};
P[388]{
   GP1:
	UF : 0, UT : 6,		CONFIG : 'N U T, 0, 0, 0',
	X =  173.893  mm,	Y =   -630.176  mm,	Z =   -253.833  mm,
	W =  90.000 deg,	P =   0.000 deg,	R =   90.000 deg
};
P[389]{
   GP1:
	UF : 0, UT : 6,		CONFIG : 'N U T, 0, 0, 0',
	X =  177.098  mm,	Y =   -628.334  mm,	Z =   -253.813  mm,
	W =  90.000 deg,	P =   0.000 deg,	R =   90.000 deg
};
P[390]{
   GP1:
	UF : 0, UT : 6,		CONFIG : 'N U T, 0, 0, 0',
	X =  178.651  mm,	Y =   -627.382  mm,	Z =   -253.947  mm,
	W =  90.000 deg,	P =   0.000 deg,	R =   90.000 deg
};
P[391]{
   GP1:
	UF : 0, UT : 6,		CONFIG : 'N U T, 0, 0, 0',
	X =  180.197  mm,	Y =   -626.528  mm,	Z =   -253.855  mm,
	W =  90.000 deg,	P =   0.000 deg,	R =   90.000 deg
};
P[392]{
   GP1:
	UF : 0, UT : 6,		CONFIG : 'N U T, 0, 0, 0',
	X =  180.887  mm,	Y =   -626.108  mm,	Z =   -253.906  mm,
	W =  90.000 deg,	P =   0.000 deg,	R =   90.000 deg
};
P[393]{
   GP1:
	UF : 0, UT : 6,		CONFIG : 'N U T, 0, 0, 0',
	X =  181.456  mm,	Y =   -625.692  mm,	Z =   -254.117  mm,
	W =  90.000 deg,	P =   0.000 deg,	R =   90.000 deg
};
P[394]{
   GP1:
	UF : 0, UT : 6,		CONFIG : 'N U T, 0, 0, 0',
	X =  182.165  mm,	Y =   -625.424  mm,	Z =   -253.772  mm,
	W =  90.000 deg,	P =   0.000 deg,	R =   90.000 deg
};
P[395]{
   GP1:
	UF : 0, UT : 6,		CONFIG : 'N U T, 0, 0, 0',
	X =  184.178  mm,	Y =   -624.237  mm,	Z =   -253.834  mm,
	W =  90.000 deg,	P =   0.000 deg,	R =   90.000 deg
};
P[396]{
   GP1:
	UF : 0, UT : 6,		CONFIG : 'N U T, 0, 0, 0',
	X =  185.737  mm,	Y =   -623.407  mm,	Z =   -253.665  mm,
	W =  90.000 deg,	P =   0.000 deg,	R =   90.000 deg
};
P[397]{
   GP1:
	UF : 0, UT : 6,		CONFIG : 'N U T, 0, 0, 0',
	X =  187.493  mm,	Y =   -622.385  mm,	Z =   -253.683  mm,
	W =  90.000 deg,	P =   0.000 deg,	R =   90.000 deg
};
P[398]{
   GP1:
	UF : 0, UT : 6,		CONFIG : 'N U T, 0, 0, 0',
	X =  188.774  mm,	Y =   -621.575  mm,	Z =   -253.856  mm,
	W =  90.000 deg,	P =   0.000 deg,	R =   90.000 deg
};
P[399]{
   GP1:
	UF : 0, UT : 6,		CONFIG : 'N U T, 0, 0, 0',
	X =  190.507  mm,	Y =   -620.610  mm,	Z =   -253.768  mm,
	W =  90.000 deg,	P =   0.000 deg,	R =   90.000 deg
};
P[400]{
   GP1:
	UF : 0, UT : 6,		CONFIG : 'N U T, 0, 0, 0',
	X =  191.557  mm,	Y =   -619.888  mm,	Z =   -254.049  mm,
	W =  90.000 deg,	P =   0.000 deg,	R =   90.000 deg
};
P[401]{
   GP1:
	UF : 0, UT : 6,		CONFIG : 'N U T, 0, 0, 0',
	X =  192.194  mm,	Y =   -619.679  mm,	Z =   -253.663  mm,
	W =  90.000 deg,	P =   0.000 deg,	R =   90.000 deg
};
P[402]{
   GP1:
	UF : 0, UT : 6,		CONFIG : 'N U T, 0, 0, 0',
	X =  193.971  mm,	Y =   -618.550  mm,	Z =   -253.914  mm,
	W =  90.000 deg,	P =   0.000 deg,	R =   90.000 deg
};
P[403]{
   GP1:
	UF : 0, UT : 6,		CONFIG : 'N U T, 0, 0, 0',
	X =  194.982  mm,	Y =   -617.974  mm,	Z =   -253.896  mm,
	W =  90.000 deg,	P =   0.000 deg,	R =   90.000 deg
};
P[404]{
   GP1:
	UF : 0, UT : 6,		CONFIG : 'N U T, 0, 0, 0',
	X =  196.361  mm,	Y =   -617.195  mm,	Z =   -253.854  mm,
	W =  90.000 deg,	P =   0.000 deg,	R =   90.000 deg
};
P[405]{
   GP1:
	UF : 0, UT : 6,		CONFIG : 'N U T, 0, 0, 0',
	X =  197.401  mm,	Y =   -616.488  mm,	Z =   -254.111  mm,
	W =  90.000 deg,	P =   0.000 deg,	R =   90.000 deg
};
P[406]{
   GP1:
	UF : 0, UT : 6,		CONFIG : 'N U T, 0, 0, 0',
	X =  198.586  mm,	Y =   -615.883  mm,	Z =   -253.918  mm,
	W =  90.000 deg,	P =   0.000 deg,	R =   90.000 deg
};
P[407]{
   GP1:
	UF : 0, UT : 6,		CONFIG : 'N U T, 0, 0, 0',
	X =  200.043  mm,	Y =   -615.098  mm,	Z =   -253.782  mm,
	W =  90.000 deg,	P =   0.000 deg,	R =   90.000 deg
};
P[408]{
   GP1:
	UF : 0, UT : 6,		CONFIG : 'N U T, 0, 0, 0',
	X =  200.867  mm,	Y =   -614.662  mm,	Z =   -253.686  mm,
	W =  90.000 deg,	P =   0.000 deg,	R =   90.000 deg
};
P[409]{
   GP1:
	UF : 0, UT : 6,		CONFIG : 'N U T, 0, 0, 0',
	X =  203.321  mm,	Y =   -613.136  mm,	Z =   -253.950  mm,
	W =  90.000 deg,	P =   0.000 deg,	R =   90.000 deg
};
P[410]{
   GP1:
	UF : 0, UT : 6,		CONFIG : 'N U T, 0, 0, 0',
	X =  204.899  mm,	Y =   -612.164  mm,	Z =   -254.098  mm,
	W =  90.000 deg,	P =   0.000 deg,	R =   90.000 deg
};
P[411]{
   GP1:
	UF : 0, UT : 6,		CONFIG : 'N U T, 0, 0, 0',
	X =  206.618  mm,	Y =   -611.234  mm,	Z =   -253.947  mm,
	W =  90.000 deg,	P =   0.000 deg,	R =   90.000 deg
};
P[412]{
   GP1:
	UF : 0, UT : 6,		CONFIG : 'N U T, 0, 0, 0',
	X =  208.390  mm,	Y =   -610.150  mm,	Z =   -254.093  mm,
	W =  90.000 deg,	P =   0.000 deg,	R =   90.000 deg
};
P[413]{
   GP1:
	UF : 0, UT : 6,		CONFIG : 'N U T, 0, 0, 0',
	X =  209.057  mm,	Y =   -609.766  mm,	Z =   -254.091  mm,
	W =  90.000 deg,	P =   0.000 deg,	R =   90.000 deg
};
P[414]{
   GP1:
	UF : 0, UT : 6,		CONFIG : 'N U T, 0, 0, 0',
	X =  210.367  mm,	Y =   -609.174  mm,	Z =   -253.692  mm,
	W =  90.000 deg,	P =   0.000 deg,	R =   90.000 deg
};
P[415]{
   GP1:
	UF : 0, UT : 6,		CONFIG : 'N U T, 0, 0, 0',
	X =  211.415  mm,	Y =   -608.428  mm,	Z =   -254.033  mm,
	W =  90.000 deg,	P =   0.000 deg,	R =   90.000 deg
};
P[416]{
   GP1:
	UF : 0, UT : 6,		CONFIG : 'N U T, 0, 0, 0',
	X =  212.531  mm,	Y =   -607.864  mm,	Z =   -253.839  mm,
	W =  90.000 deg,	P =   0.000 deg,	R =   90.000 deg
};
P[417]{
   GP1:
	UF : 0, UT : 6,		CONFIG : 'N U T, 0, 0, 0',
	X =  216.353  mm,	Y =   -605.647  mm,	Z =   -253.865  mm,
	W =  90.000 deg,	P =   0.000 deg,	R =   90.000 deg
};
P[418]{
   GP1:
	UF : 0, UT : 6,		CONFIG : 'N U T, 0, 0, 0',
	X =  217.171  mm,	Y =   -605.129  mm,	Z =   -253.976  mm,
	W =  90.000 deg,	P =   0.000 deg,	R =   90.000 deg
};
P[419]{
   GP1:
	UF : 0, UT : 6,		CONFIG : 'N U T, 0, 0, 0',
	X =  220.039  mm,	Y =   -603.422  mm,	Z =   -254.099  mm,
	W =  90.000 deg,	P =   0.000 deg,	R =   90.000 deg
};
P[420]{
   GP1:
	UF : 0, UT : 6,		CONFIG : 'N U T, 0, 0, 0',
	X =  222.534  mm,	Y =   -601.991  mm,	Z =   -254.077  mm,
	W =  90.000 deg,	P =   0.000 deg,	R =   90.000 deg
};
P[421]{
   GP1:
	UF : 0, UT : 6,		CONFIG : 'N U T, 0, 0, 0',
	X =  223.322  mm,	Y =   -601.645  mm,	Z =   -253.810  mm,
	W =  90.000 deg,	P =   0.000 deg,	R =   90.000 deg
};
P[422]{
   GP1:
	UF : 0, UT : 6,		CONFIG : 'N U T, 0, 0, 0',
	X =  226.177  mm,	Y =   -599.995  mm,	Z =   -253.815  mm,
	W =  90.000 deg,	P =   0.000 deg,	R =   90.000 deg
};
P[423]{
   GP1:
	UF : 0, UT : 6,		CONFIG : 'N U T, 0, 0, 0',
	X =  230.315  mm,	Y =   -597.495  mm,	Z =   -254.084  mm,
	W =  90.000 deg,	P =   0.000 deg,	R =   90.000 deg
};
P[424]{
   GP1:
	UF : 0, UT : 6,		CONFIG : 'N U T, 0, 0, 0',
	X =  233.160  mm,	Y =   -595.945  mm,	Z =   -253.857  mm,
	W =  90.000 deg,	P =   0.000 deg,	R =   90.000 deg
};
P[425]{
   GP1:
	UF : 0, UT : 6,		CONFIG : 'N U T, 0, 0, 0',
	X =  233.779  mm,	Y =   -595.666  mm,	Z =   -253.669  mm,
	W =  90.000 deg,	P =   0.000 deg,	R =   90.000 deg
};
P[426]{
   GP1:
	UF : 0, UT : 6,		CONFIG : 'N U T, 0, 0, 0',
	X =  235.720  mm,	Y =   -594.384  mm,	Z =   -254.058  mm,
	W =  90.000 deg,	P =   0.000 deg,	R =   90.000 deg
};
P[427]{
   GP1:
	UF : 0, UT : 6,		CONFIG : 'N U T, 0, 0, 0',
	X =  239.909  mm,	Y =   -592.111  mm,	Z =   -253.707  mm,
	W =  90.000 deg,	P =   0.000 deg,	R =   90.000 deg
};
P[428]{
   GP1:
	UF : 0, UT : 6,		CONFIG : 'N U T, 0, 0, 0',
	X =  240.586  mm,	Y =   -591.645  mm,	Z =   -253.890  mm,
	W =  90.000 deg,	P =   0.000 deg,	R =   90.000 deg
};
P[429]{
   GP1:
	UF : 0, UT : 6,		CONFIG : 'N U T, 0, 0, 0',
	X =  241.630  mm,	Y =   -591.052  mm,	Z =   -253.864  mm,
	W =  90.000 deg,	P =   0.000 deg,	R =   90.000 deg
};
P[430]{
   GP1:
	UF : 0, UT : 6,		CONFIG : 'N U T, 0, 0, 0',
	X =  243.410  mm,	Y =   -590.078  mm,	Z =   -253.734  mm,
	W =  90.000 deg,	P =   0.000 deg,	R =   90.000 deg
};
P[431]{
   GP1:
	UF : 0, UT : 6,		CONFIG : 'N U T, 0, 0, 0',
	X =  244.625  mm,	Y =   -589.217  mm,	Z =   -254.121  mm,
	W =  90.000 deg,	P =   0.000 deg,	R =   90.000 deg
};
P[432]{
   GP1:
	UF : 0, UT : 6,		CONFIG : 'N U T, 0, 0, 0',
	X =  247.372  mm,	Y =   -587.776  mm,	Z =   -253.768  mm,
	W =  90.000 deg,	P =   0.000 deg,	R =   90.000 deg
};
P[433]{
   GP1:
	UF : 0, UT : 6,		CONFIG : 'N U T, 0, 0, 0',
	X =  249.854  mm,	Y =   -586.285  mm,	Z =   -253.910  mm,
	W =  90.000 deg,	P =   0.000 deg,	R =   90.000 deg
};
P[434]{
   GP1:
	UF : 0, UT : 6,		CONFIG : 'N U T, 0, 0, 0',
	X =  252.767  mm,	Y =   -584.575  mm,	Z =   -253.975  mm,
	W =  90.000 deg,	P =   0.000 deg,	R =   90.000 deg
};
P[435]{
   GP1:
	UF : 0, UT : 6,		CONFIG : 'N U T, 0, 0, 0',
	X =  256.146  mm,	Y =   -582.657  mm,	Z =   -253.897  mm,
	W =  90.000 deg,	P =   0.000 deg,	R =   90.000 deg
};
P[436]{
   GP1:
	UF : 0, UT : 6,		CONFIG : 'N U T, 0, 0, 0',
	X =  256.773  mm,	Y =   -582.393  mm,	Z =   -253.661  mm,
	W =  90.000 deg,	P =   0.000 deg,	R =   90.000 deg
};
P[437]{
   GP1:
	UF : 0, UT : 6,		CONFIG : 'N U T, 0, 0, 0',
	X =  260.094  mm,	Y =   -580.358  mm,	Z =   -253.944  mm,
	W =  90.000 deg,	P =   0.000 deg,	R =   90.000 deg
};
P[438]{
   GP1:
	UF : 0, UT : 6,		CONFIG : 'N U T, 0, 0, 0',
	X =  261.050  mm,	Y =   -579.846  mm,	Z =   -253.849  mm,
	W =  90.000 deg,	P =   0.000 deg,	R =   90.000 deg
};
P[439]{
   GP1:
	UF : 0, UT : 6,		CONFIG : 'N U T, 0, 0, 0',
	X =  262.708  mm,	Y =   -578.893  mm,	Z =   -253.836  mm,
	W =  90.000 deg,	P =   0.000 deg,	R =   90.000 deg
};
P[440]{
   GP1:
	UF : 0, UT : 6,		CONFIG : 'N U T, 0, 0, 0',
	X =  263.927  mm,	Y =   -578.207  mm,	Z =   -253.795  mm,
	W =  90.000 deg,	P =   0.000 deg,	R =   90.000 deg
};
P[441]{
   GP1:
	UF : 0, UT : 6,		CONFIG : 'N U T, 0, 0, 0',
	X =  265.115  mm,	Y =   -577.452  mm,	Z =   -253.964  mm,
	W =  90.000 deg,	P =   0.000 deg,	R =   90.000 deg
};
P[442]{
   GP1:
	UF : 0, UT : 6,		CONFIG : 'N U T, 0, 0, 0',
	X =  265.815  mm,	Y =   -577.128  mm,	Z =   -253.767  mm,
	W =  90.000 deg,	P =   0.000 deg,	R =   90.000 deg
};
P[443]{
   GP1:
	UF : 0, UT : 6,		CONFIG : 'N U T, 0, 0, 0',
	X =  266.400  mm,	Y =   -576.646  mm,	Z =   -254.119  mm,
	W =  90.000 deg,	P =   0.000 deg,	R =   90.000 deg
};
P[444]{
   GP1:
	UF : 0, UT : 6,		CONFIG : 'N U T, 0, 0, 0',
	X =  269.651  mm,	Y =   -574.901  mm,	Z =   -253.796  mm,
	W =  90.000 deg,	P =   0.000 deg,	R =   90.000 deg
};
P[445]{
   GP1:
	UF : 0, UT : 6,		CONFIG : 'N U T, 0, 0, 0',
	X =  270.217  mm,	Y =   -574.487  mm,	Z =   -254.009  mm,
	W =  90.000 deg,	P =   0.000 deg,	R =   90.000 deg
};
P[446]{
   GP1:
	UF : 0, UT : 6,		CONFIG : 'N U T, 0, 0, 0',
	X =  270.803  mm,	Y =   -574.109  mm,	Z =   -254.105  mm,
	W =  90.000 deg,	P =   0.000 deg,	R =   90.000 deg
};
P[447]{
   GP1:
	UF : 0, UT : 6,		CONFIG : 'N U T, 0, 0, 0',
	X =  271.415  mm,	Y =   -573.808  mm,	Z =   -253.978  mm,
	W =  90.000 deg,	P =   0.000 deg,	R =   90.000 deg
};
P[448]{
   GP1:
	UF : 0, UT : 6,		CONFIG : 'N U T, 0, 0, 0',
	X =  272.339  mm,	Y =   -573.365  mm,	Z =   -253.756  mm,
	W =  90.000 deg,	P =   0.000 deg,	R =   90.000 deg
};
P[449]{
   GP1:
	UF : 0, UT : 6,		CONFIG : 'N U T, 0, 0, 0',
	X =  273.762  mm,	Y =   -572.490  mm,	Z =   -253.887  mm,
	W =  90.000 deg,	P =   0.000 deg,	R =   90.000 deg
};
P[450]{
   GP1:
	UF : 0, UT : 6,		CONFIG : 'N U T, 0, 0, 0',
	X =  278.571  mm,	Y =   -569.728  mm,	Z =   -253.852  mm,
	W =  90.000 deg,	P =   0.000 deg,	R =   90.000 deg
};
P[451]{
   GP1:
	UF : 0, UT : 6,		CONFIG : 'N U T, 0, 0, 0',
	X =  281.293  mm,	Y =   -568.187  mm,	Z =   -253.775  mm,
	W =  90.000 deg,	P =   0.000 deg,	R =   90.000 deg
};
P[452]{
   GP1:
	UF : 0, UT : 6,		CONFIG : 'N U T, 0, 0, 0',
	X =  285.461  mm,	Y =   -565.772  mm,	Z =   -253.796  mm,
	W =  90.000 deg,	P =   0.000 deg,	R =   90.000 deg
};
P[453]{
   GP1:
	UF : 0, UT : 6,		CONFIG : 'N U T, 0, 0, 0',
	X =  291.269  mm,	Y =   -562.325  mm,	Z =   -254.027  mm,
	W =  90.000 deg,	P =   0.000 deg,	R =   90.000 deg
};
P[454]{
   GP1:
	UF : 0, UT : 6,		CONFIG : 'N U T, 0, 0, 0',
	X =  292.384  mm,	Y =   -561.793  mm,	Z =   -253.754  mm,
	W =  90.000 deg,	P =   0.000 deg,	R =   90.000 deg
};
P[455]{
   GP1:
	UF : 0, UT : 6,		CONFIG : 'N U T, 0, 0, 0',
	X =  294.243  mm,	Y =   -560.711  mm,	Z =   -253.773  mm,
	W =  90.000 deg,	P =   0.000 deg,	R =   90.000 deg
};
P[456]{
   GP1:
	UF : 0, UT : 6,		CONFIG : 'N U T, 0, 0, 0',
	X =  295.278  mm,	Y =   -560.148  mm,	Z =   -253.691  mm,
	W =  90.000 deg,	P =   0.000 deg,	R =   90.000 deg
};
P[457]{
   GP1:
	UF : 0, UT : 6,		CONFIG : 'N U T, 0, 0, 0',
	X =  296.445  mm,	Y =   -559.434  mm,	Z =   -253.788  mm,
	W =  90.000 deg,	P =   0.000 deg,	R =   90.000 deg
};
P[458]{
   GP1:
	UF : 0, UT : 6,		CONFIG : 'N U T, 0, 0, 0',
	X =  298.346  mm,	Y =   -558.321  mm,	Z =   -253.826  mm,
	W =  90.000 deg,	P =   0.000 deg,	R =   90.000 deg
};
P[459]{
   GP1:
	UF : 0, UT : 6,		CONFIG : 'N U T, 0, 0, 0',
	X =  299.731  mm,	Y =   -557.471  mm,	Z =   -253.947  mm,
	W =  90.000 deg,	P =   0.000 deg,	R =   90.000 deg
};
P[460]{
   GP1:
	UF : 0, UT : 6,		CONFIG : 'N U T, 0, 0, 0',
	X =  301.797  mm,	Y =   -556.232  mm,	Z =   -254.058  mm,
	W =  90.000 deg,	P =   0.000 deg,	R =   90.000 deg
};
P[461]{
   GP1:
	UF : 0, UT : 6,		CONFIG : 'N U T, 0, 0, 0',
	X =  302.539  mm,	Y =   -555.790  mm,	Z =   -254.093  mm,
	W =  90.000 deg,	P =   0.000 deg,	R =   90.000 deg
};
P[462]{
   GP1:
	UF : 0, UT : 6,		CONFIG : 'N U T, 0, 0, 0',
	X =  303.569  mm,	Y =   -555.306  mm,	Z =   -253.822  mm,
	W =  90.000 deg,	P =   0.000 deg,	R =   90.000 deg
};
P[463]{
   GP1:
	UF : 0, UT : 6,		CONFIG : 'N U T, 0, 0, 0',
	X =  304.333  mm,	Y =   -554.832  mm,	Z =   -253.901  mm,
	W =  90.000 deg,	P =   0.000 deg,	R =   90.000 deg
};
P[464]{
   GP1:
	UF : 0, UT : 6,		CONFIG : 'N U T, 0, 0, 0',
	X =  305.483  mm,	Y =   -554.100  mm,	Z =   -254.068  mm,
	W =  90.000 deg,	P =   0.000 deg,	R =   90.000 deg
};
P[465]{
   GP1:
	UF : 0, UT : 6,		CONFIG : 'N U T, 0, 0, 0',
	X =  306.646  mm,	Y =   -553.576  mm,	Z =   -253.711  mm,
	W =  90.000 deg,	P =   0.000 deg,	R =   90.000 deg
};
P[466]{
   GP1:
	UF : 0, UT : 6,		CONFIG : 'N U T, 0, 0, 0',
	X =  307.241  mm,	Y =   -553.234  mm,	Z =   -253.705  mm,
	W =  90.000 deg,	P =   0.000 deg,	R =   90.000 deg
};
P[467]{
   GP1:
	UF : 0, UT : 6,		CONFIG : 'N U T, 0, 0, 0',
	X =  308.121  mm,	Y =   -552.687  mm,	Z =   -253.800  mm,
	W =  90.000 deg,	P =   0.000 deg,	R =   90.000 deg
};
P[468]{
   GP1:
	UF : 0, UT : 6,		CONFIG : 'N U T, 0, 0, 0',
	X =  309.234  mm,	Y =   -552.099  mm,	Z =   -253.668  mm,
	W =  90.000 deg,	P =   0.000 deg,	R =   90.000 deg
};
P[469]{
   GP1:
	UF : 0, UT : 6,		CONFIG : 'N U T, 0, 0, 0',
	X =  313.120  mm,	Y =   -549.845  mm,	Z =   -253.693  mm,
	W =  90.000 deg,	P =   0.000 deg,	R =   90.000 deg
};
P[470]{
   GP1:
	UF : 0, UT : 6,		CONFIG : 'N U T, 0, 0, 0',
	X =  314.195  mm,	Y =   -549.166  mm,	Z =   -253.835  mm,
	W =  90.000 deg,	P =   0.000 deg,	R =   90.000 deg
};
P[471]{
   GP1:
	UF : 0, UT : 6,		CONFIG : 'N U T, 0, 0, 0',
	X =  315.971  mm,	Y =   -548.069  mm,	Z =   -254.007  mm,
	W =  90.000 deg,	P =   0.000 deg,	R =   90.000 deg
};
P[472]{
   GP1:
	UF : 0, UT : 6,		CONFIG : 'N U T, 0, 0, 0',
	X =  322.768  mm,	Y =   -544.206  mm,	Z =   -253.859  mm,
	W =  90.000 deg,	P =   0.000 deg,	R =   90.000 deg
};
P[473]{
   GP1:
	UF : 0, UT : 6,		CONFIG : 'N U T, 0, 0, 0',
	X =  323.440  mm,	Y =   -543.839  mm,	Z =   -253.809  mm,
	W =  90.000 deg,	P =   0.000 deg,	R =   90.000 deg
};
P[474]{
   GP1:
	UF : 0, UT : 6,		CONFIG : 'N U T, 0, 0, 0',
	X =  324.242  mm,	Y =   -543.375  mm,	Z =   -253.810  mm,
	W =  90.000 deg,	P =   0.000 deg,	R =   90.000 deg
};
P[475]{
   GP1:
	UF : 0, UT : 6,		CONFIG : 'N U T, 0, 0, 0',
	X =  325.815  mm,	Y =   -542.408  mm,	Z =   -253.955  mm,
	W =  90.000 deg,	P =   0.000 deg,	R =   90.000 deg
};
P[476]{
   GP1:
	UF : 0, UT : 6,		CONFIG : 'N U T, 0, 0, 0',
	X =  326.905  mm,	Y =   -541.803  mm,	Z =   -253.895  mm,
	W =  90.000 deg,	P =   0.000 deg,	R =   90.000 deg
};
P[477]{
   GP1:
	UF : 0, UT : 6,		CONFIG : 'N U T, 0, 0, 0',
	X =  330.375  mm,	Y =   -539.855  mm,	Z =   -253.759  mm,
	W =  90.000 deg,	P =   0.000 deg,	R =   90.000 deg
};
P[478]{
   GP1:
	UF : 0, UT : 6,		CONFIG : 'N U T, 0, 0, 0',
	X =  330.987  mm,	Y =   -539.490  mm,	Z =   -253.787  mm,
	W =  90.000 deg,	P =   0.000 deg,	R =   90.000 deg
};
P[479]{
   GP1:
	UF : 0, UT : 6,		CONFIG : 'N U T, 0, 0, 0',
	X =  331.746  mm,	Y =   -538.981  mm,	Z =   -253.961  mm,
	W =  90.000 deg,	P =   0.000 deg,	R =   90.000 deg
};
P[480]{
   GP1:
	UF : 0, UT : 6,		CONFIG : 'N U T, 0, 0, 0',
	X =  333.932  mm,	Y =   -537.743  mm,	Z =   -253.901  mm,
	W =  90.000 deg,	P =   0.000 deg,	R =   90.000 deg
};
P[481]{
   GP1:
	UF : 0, UT : 6,		CONFIG : 'N U T, 0, 0, 0',
	X =  337.226  mm,	Y =   -535.896  mm,	Z =   -253.767  mm,
	W =  90.000 deg,	P =   0.000 deg,	R =   90.000 deg
};
P[482]{
   GP1:
	UF : 0, UT : 6,		CONFIG : 'N U T, 0, 0, 0',
	X =  338.247  mm,	Y =   -535.253  mm,	Z =   -253.898  mm,
	W =  90.000 deg,	P =   0.000 deg,	R =   90.000 deg
};
P[483]{
   GP1:
	UF : 0, UT : 6,		CONFIG : 'N U T, 0, 0, 0',
	X =  340.097  mm,	Y =   -534.256  mm,	Z =   -253.723  mm,
	W =  90.000 deg,	P =   0.000 deg,	R =   90.000 deg
};
P[484]{
   GP1:
	UF : 0, UT : 6,		CONFIG : 'N U T, 0, 0, 0',
	X =  341.454  mm,	Y =   -533.401  mm,	Z =   -253.897  mm,
	W =  90.000 deg,	P =   0.000 deg,	R =   90.000 deg
};
P[485]{
   GP1:
	UF : 0, UT : 6,		CONFIG : 'N U T, 0, 0, 0',
	X =  344.712  mm,	Y =   -531.503  mm,	Z =   -253.938  mm,
	W =  90.000 deg,	P =   0.000 deg,	R =   90.000 deg
};
P[486]{
   GP1:
	UF : 0, UT : 6,		CONFIG : 'N U T, 0, 0, 0',
	X =  345.626  mm,	Y =   -530.912  mm,	Z =   -254.091  mm,
	W =  90.000 deg,	P =   0.000 deg,	R =   90.000 deg
};
P[487]{
   GP1:
	UF : 0, UT : 6,		CONFIG : 'N U T, 0, 0, 0',
	X =  347.246  mm,	Y =   -530.128  mm,	Z =   -253.724  mm,
	W =  90.000 deg,	P =   0.000 deg,	R =   90.000 deg
};
P[488]{
   GP1:
	UF : 0, UT : 6,		CONFIG : 'N U T, 0, 0, 0',
	X =  350.229  mm,	Y =   -528.382  mm,	Z =   -253.783  mm,
	W =  90.000 deg,	P =   0.000 deg,	R =   90.000 deg
};
P[489]{
   GP1:
	UF : 0, UT : 6,		CONFIG : 'N U T, 0, 0, 0',
	X =  350.917  mm,	Y =   -527.909  mm,	Z =   -253.964  mm,
	W =  90.000 deg,	P =   0.000 deg,	R =   90.000 deg
};
P[490]{
   GP1:
	UF : 0, UT : 6,		CONFIG : 'N U T, 0, 0, 0',
	X =  351.899  mm,	Y =   -527.399  mm,	Z =   -253.828  mm,
	W =  90.000 deg,	P =   0.000 deg,	R =   90.000 deg
};
P[491]{
   GP1:
	UF : 0, UT : 6,		CONFIG : 'N U T, 0, 0, 0',
	X =  352.589  mm,	Y =   -526.892  mm,	Z =   -254.092  mm,
	W =  90.000 deg,	P =   0.000 deg,	R =   90.000 deg
};
P[492]{
   GP1:
	UF : 0, UT : 6,		CONFIG : 'N U T, 0, 0, 0',
	X =  353.300  mm,	Y =   -526.578  mm,	Z =   -253.859  mm,
	W =  90.000 deg,	P =   0.000 deg,	R =   90.000 deg
};
P[493]{
   GP1:
	UF : 0, UT : 6,		CONFIG : 'N U T, 0, 0, 0',
	X =  355.484  mm,	Y =   -525.302  mm,	Z =   -253.893  mm,
	W =  90.000 deg,	P =   0.000 deg,	R =   90.000 deg
};
P[494]{
   GP1:
	UF : 0, UT : 6,		CONFIG : 'N U T, 0, 0, 0',
	X =  358.165  mm,	Y =   -523.743  mm,	Z =   -253.919  mm,
	W =  90.000 deg,	P =   0.000 deg,	R =   90.000 deg
};
P[495]{
   GP1:
	UF : 0, UT : 6,		CONFIG : 'N U T, 0, 0, 0',
	X =  358.829  mm,	Y =   -523.326  mm,	Z =   -254.001  mm,
	W =  90.000 deg,	P =   0.000 deg,	R =   90.000 deg
};
P[496]{
   GP1:
	UF : 0, UT : 6,		CONFIG : 'N U T, 0, 0, 0',
	X =  359.531  mm,	Y =   -522.871  mm,	Z =   -254.123  mm,
	W =  90.000 deg,	P =   0.000 deg,	R =   90.000 deg
};
P[497]{
   GP1:
	UF : 0, UT : 6,		CONFIG : 'N U T, 0, 0, 0',
	X =  361.246  mm,	Y =   -522.002  mm,	Z =   -253.829  mm,
	W =  90.000 deg,	P =   0.000 deg,	R =   90.000 deg
};
P[498]{
   GP1:
	UF : 0, UT : 6,		CONFIG : 'N U T, 0, 0, 0',
	X =  365.900  mm,	Y =   -519.361  mm,	Z =   -253.716  mm,
	W =  90.000 deg,	P =   0.000 deg,	R =   90.000 deg
};
P[499]{
   GP1:
	UF : 0, UT : 6,		CONFIG : 'N U T, 0, 0, 0',
	X =  367.089  mm,	Y =   -518.539  mm,	Z =   -254.045  mm,
	W =  90.000 deg,	P =   0.000 deg,	R =   90.000 deg
};
P[500]{
   GP1:
	UF : 0, UT : 6,		CONFIG : 'N U T, 0, 0, 0',
	X =  368.616  mm,	Y =   -517.673  mm,	Z =   -254.006  mm,
	W =  90.000 deg,	P =   0.000 deg,	R =   90.000 deg
};
P[501]{
   GP1:
	UF : 0, UT : 6,		CONFIG : 'N U T, 0, 0, 0',
	X =  370.166  mm,	Y =   -516.850  mm,	Z =   -253.832  mm,
	W =  90.000 deg,	P =   0.000 deg,	R =   90.000 deg
};
P[502]{
   GP1:
	UF : 0, UT : 6,		CONFIG : 'N U T, 0, 0, 0',
	X =  371.883  mm,	Y =   -515.876  mm,	Z =   -253.791  mm,
	W =  90.000 deg,	P =   0.000 deg,	R =   90.000 deg
};
P[503]{
   GP1:
	UF : 0, UT : 6,		CONFIG : 'N U T, 0, 0, 0',
	X =  372.493  mm,	Y =   -515.400  mm,	Z =   -254.093  mm,
	W =  90.000 deg,	P =   0.000 deg,	R =   90.000 deg
};
P[504]{
   GP1:
	UF : 0, UT : 6,		CONFIG : 'N U T, 0, 0, 0',
	X =  373.735  mm,	Y =   -514.703  mm,	Z =   -254.042  mm,
	W =  90.000 deg,	P =   0.000 deg,	R =   90.000 deg
};
P[505]{
   GP1:
	UF : 0, UT : 6,		CONFIG : 'N U T, 0, 0, 0',
	X =  374.422  mm,	Y =   -514.441  mm,	Z =   -253.715  mm,
	W =  90.000 deg,	P =   0.000 deg,	R =   90.000 deg
};
P[506]{
   GP1:
	UF : 0, UT : 6,		CONFIG : 'N U T, 0, 0, 0',
	X =  375.541  mm,	Y =   -513.810  mm,	Z =   -253.677  mm,
	W =  90.000 deg,	P =   0.000 deg,	R =   90.000 deg
};
P[507]{
   GP1:
	UF : 0, UT : 6,		CONFIG : 'N U T, 0, 0, 0',
	X =  382.246  mm,	Y =   -509.795  mm,	Z =   -254.025  mm,
	W =  90.000 deg,	P =   0.000 deg,	R =   90.000 deg
};
P[508]{
   GP1:
	UF : 0, UT : 6,		CONFIG : 'N U T, 0, 0, 0',
	X =  383.574  mm,	Y =   -509.102  mm,	Z =   -253.849  mm,
	W =  90.000 deg,	P =   0.000 deg,	R =   90.000 deg
};
P[509]{
   GP1:
	UF : 0, UT : 6,		CONFIG : 'N U T, 0, 0, 0',
	X =  384.642  mm,	Y =   -508.532  mm,	Z =   -253.734  mm,
	W =  90.000 deg,	P =   0.000 deg,	R =   90.000 deg
};
P[510]{
   GP1:
	UF : 0, UT : 6,		CONFIG : 'N U T, 0, 0, 0',
	X =  385.623  mm,	Y =   -507.807  mm,	Z =   -254.121  mm,
	W =  90.000 deg,	P =   0.000 deg,	R =   90.000 deg
};
P[511]{
   GP1:
	UF : 0, UT : 6,		CONFIG : 'N U T, 0, 0, 0',
	X =  386.670  mm,	Y =   -507.202  mm,	Z =   -254.119  mm,
	W =  90.000 deg,	P =   0.000 deg,	R =   90.000 deg
};
P[512]{
   GP1:
	UF : 0, UT : 6,		CONFIG : 'N U T, 0, 0, 0',
	X =  387.969  mm,	Y =   -506.564  mm,	Z =   -253.849  mm,
	W =  90.000 deg,	P =   0.000 deg,	R =   90.000 deg
};
P[513]{
   GP1:
	UF : 0, UT : 6,		CONFIG : 'N U T, 0, 0, 0',
	X =  389.270  mm,	Y =   -505.861  mm,	Z =   -253.734  mm,
	W =  90.000 deg,	P =   0.000 deg,	R =   90.000 deg
};
P[514]{
   GP1:
	UF : 0, UT : 6,		CONFIG : 'N U T, 0, 0, 0',
	X =  390.587  mm,	Y =   -505.042  mm,	Z =   -253.874  mm,
	W =  90.000 deg,	P =   0.000 deg,	R =   90.000 deg
};
P[515]{
   GP1:
	UF : 0, UT : 6,		CONFIG : 'N U T, 0, 0, 0',
	X =  391.202  mm,	Y =   -504.681  mm,	Z =   -253.890  mm,
	W =  90.000 deg,	P =   0.000 deg,	R =   90.000 deg
};
P[516]{
   GP1:
	UF : 0, UT : 6,		CONFIG : 'N U T, 0, 0, 0',
	X =  396.819  mm,	Y =   -501.423  mm,	Z =   -253.925  mm,
	W =  90.000 deg,	P =   0.000 deg,	R =   90.000 deg
};
P[517]{
   GP1:
	UF : 0, UT : 6,		CONFIG : 'N U T, 0, 0, 0',
	X =  398.402  mm,	Y =   -500.533  mm,	Z =   -253.864  mm,
	W =  90.000 deg,	P =   0.000 deg,	R =   90.000 deg
};
P[518]{
   GP1:
	UF : 0, UT : 6,		CONFIG : 'N U T, 0, 0, 0',
	X =  399.129  mm,	Y =   -500.027  mm,	Z =   -254.075  mm,
	W =  90.000 deg,	P =   0.000 deg,	R =   90.000 deg
};
P[519]{
   GP1:
	UF : 0, UT : 6,		CONFIG : 'N U T, 0, 0, 0',
	X =  400.344  mm,	Y =   -499.441  mm,	Z =   -253.796  mm,
	W =  90.000 deg,	P =   0.000 deg,	R =   90.000 deg
};
P[520]{
   GP1:
	UF : 0, UT : 6,		CONFIG : 'N U T, 0, 0, 0',
	X =  404.024  mm,	Y =   -497.191  mm,	Z =   -254.097  mm,
	W =  90.000 deg,	P =   0.000 deg,	R =   90.000 deg
};
P[521]{
   GP1:
	UF : 0, UT : 6,		CONFIG : 'N U T, 0, 0, 0',
	X =  405.765  mm,	Y =   -496.230  mm,	Z =   -253.990  mm,
	W =  90.000 deg,	P =   0.000 deg,	R =   90.000 deg
};
P[522]{
   GP1:
	UF : 0, UT : 6,		CONFIG : 'N U T, 0, 0, 0',
	X =  406.485  mm,	Y =   -495.807  mm,	Z =   -254.008  mm,
	W =  90.000 deg,	P =   0.000 deg,	R =   90.000 deg
};
P[523]{
   GP1:
	UF : 0, UT : 6,		CONFIG : 'N U T, 0, 0, 0',
	X =  408.586  mm,	Y =   -494.546  mm,	Z =   -254.126  mm,
	W =  90.000 deg,	P =   0.000 deg,	R =   90.000 deg
};
P[524]{
   GP1:
	UF : 0, UT : 6,		CONFIG : 'N U T, 0, 0, 0',
	X =  409.496  mm,	Y =   -494.165  mm,	Z =   -253.773  mm,
	W =  90.000 deg,	P =   0.000 deg,	R =   90.000 deg
};
P[525]{
   GP1:
	UF : 0, UT : 6,		CONFIG : 'N U T, 0, 0, 0',
	X =  410.928  mm,	Y =   -493.389  mm,	Z =   -253.651  mm,
	W =  90.000 deg,	P =   0.000 deg,	R =   90.000 deg
};
P[526]{
   GP1:
	UF : 0, UT : 6,		CONFIG : 'N U T, 0, 0, 0',
	X =  411.859  mm,	Y =   -492.850  mm,	Z =   -253.655  mm,
	W =  90.000 deg,	P =   0.000 deg,	R =   90.000 deg
};
P[527]{
   GP1:
	UF : 0, UT : 6,		CONFIG : 'N U T, 0, 0, 0',
	X =  413.245  mm,	Y =   -491.856  mm,	Z =   -254.124  mm,
	W =  90.000 deg,	P =   0.000 deg,	R =   90.000 deg
};
P[528]{
   GP1:
	UF : 0, UT : 6,		CONFIG : 'N U T, 0, 0, 0',
	X =  416.894  mm,	Y =   -489.862  mm,	Z =   -253.852  mm,
	W =  90.000 deg,	P =   0.000 deg,	R =   90.000 deg
};
P[529]{
   GP1:
	UF : 0, UT : 6,		CONFIG : 'N U T, 0, 0, 0',
	X =  418.529  mm,	Y =   -488.997  mm,	Z =   -253.658  mm,
	W =  90.000 deg,	P =   0.000 deg,	R =   90.000 deg
};
P[530]{
   GP1:
	UF : 0, UT : 6,		CONFIG : 'N U T, 0, 0, 0',
	X =  419.558  mm,	Y =   -488.355  mm,	Z =   -253.775  mm,
	W =  90.000 deg,	P =   0.000 deg,	R =   90.000 deg
};
P[531]{
   GP1:
	UF : 0, UT : 6,		CONFIG : 'N U T, 0, 0, 0',
	X =  420.601  mm,	Y =   -487.742  mm,	Z =   -253.800  mm,
	W =  90.000 deg,	P =   0.000 deg,	R =   90.000 deg
};
P[532]{
   GP1:
	UF : 0, UT : 6,		CONFIG : 'N U T, 0, 0, 0',
	X =  422.790  mm,	Y =   -486.399  mm,	Z =   -253.993  mm,
	W =  90.000 deg,	P =   0.000 deg,	R =   90.000 deg
};
P[533]{
   GP1:
	UF : 0, UT : 6,		CONFIG : 'N U T, 0, 0, 0',
	X =  423.458  mm,	Y =   -486.010  mm,	Z =   -254.000  mm,
	W =  90.000 deg,	P =   0.000 deg,	R =   90.000 deg
};
P[534]{
   GP1:
	UF : 0, UT : 6,		CONFIG : 'N U T, 0, 0, 0',
	X =  424.408  mm,	Y =   -485.594  mm,	Z =   -253.679  mm,
	W =  90.000 deg,	P =   0.000 deg,	R =   90.000 deg
};
P[535]{
   GP1:
	UF : 0, UT : 6,		CONFIG : 'N U T, 0, 0, 0',
	X =  426.183  mm,	Y =   -484.456  mm,	Z =   -253.954  mm,
	W =  90.000 deg,	P =   0.000 deg,	R =   90.000 deg
};
P[536]{
   GP1:
	UF : 0, UT : 6,		CONFIG : 'N U T, 0, 0, 0',
	X =  426.939  mm,	Y =   -484.094  mm,	Z =   -253.773  mm,
	W =  90.000 deg,	P =   0.000 deg,	R =   90.000 deg
};
P[537]{
   GP1:
	UF : 0, UT : 6,		CONFIG : 'N U T, 0, 0, 0',
	X =  428.277  mm,	Y =   -483.330  mm,	Z =   -253.752  mm,
	W =  90.000 deg,	P =   0.000 deg,	R =   90.000 deg
};
P[538]{
   GP1:
	UF : 0, UT : 6,		CONFIG : 'N U T, 0, 0, 0',
	X =  430.602  mm,	Y =   -481.842  mm,	Z =   -254.106  mm,
	W =  90.000 deg,	P =   0.000 deg,	R =   90.000 deg
};
P[539]{
   GP1:
	UF : 0, UT : 6,		CONFIG : 'N U T, 0, 0, 0',
	X =  431.237  mm,	Y =   -481.644  mm,	Z =   -253.696  mm,
	W =  90.000 deg,	P =   0.000 deg,	R =   90.000 deg
};
P[540]{
   GP1:
	UF : 0, UT : 6,		CONFIG : 'N U T, 0, 0, 0',
	X =  432.108  mm,	Y =   -481.068  mm,	Z =   -253.876  mm,
	W =  90.000 deg,	P =   0.000 deg,	R =   90.000 deg
};
P[541]{
   GP1:
	UF : 0, UT : 6,		CONFIG : 'N U T, 0, 0, 0',
	X =  433.144  mm,	Y =   -480.402  mm,	Z =   -254.039  mm,
	W =  90.000 deg,	P =   0.000 deg,	R =   90.000 deg
};
P[542]{
   GP1:
	UF : 0, UT : 6,		CONFIG : 'N U T, 0, 0, 0',
	X =  434.230  mm,	Y =   -479.753  mm,	Z =   -254.091  mm,
	W =  90.000 deg,	P =   0.000 deg,	R =   90.000 deg
};
P[543]{
   GP1:
	UF : 0, UT : 6,		CONFIG : 'N U T, 0, 0, 0',
	X =  437.690  mm,	Y =   -477.743  mm,	Z =   -254.123  mm,
	W =  90.000 deg,	P =   0.000 deg,	R =   90.000 deg
};
P[544]{
   GP1:
	UF : 0, UT : 6,		CONFIG : 'N U T, 0, 0, 0',
	X =  439.027  mm,	Y =   -477.097  mm,	Z =   -253.814  mm,
	W =  90.000 deg,	P =   0.000 deg,	R =   90.000 deg
};
P[545]{
   GP1:
	UF : 0, UT : 6,		CONFIG : 'N U T, 0, 0, 0',
	X =  440.811  mm,	Y =   -476.027  mm,	Z =   -253.914  mm,
	W =  90.000 deg,	P =   0.000 deg,	R =   90.000 deg
};
P[546]{
   GP1:
	UF : 0, UT : 6,		CONFIG : 'N U T, 0, 0, 0',
	X =  443.077  mm,	Y =   -474.782  mm,	Z =   -253.760  mm,
	W =  90.000 deg,	P =   0.000 deg,	R =   90.000 deg
};
P[547]{
   GP1:
	UF : 0, UT : 6,		CONFIG : 'N U T, 0, 0, 0',
	X =  444.486  mm,	Y =   -473.984  mm,	Z =   -253.722  mm,
	W =  90.000 deg,	P =   0.000 deg,	R =   90.000 deg
};
P[548]{
   GP1:
	UF : 0, UT : 6,		CONFIG : 'N U T, 0, 0, 0',
	X =  446.819  mm,	Y =   -472.621  mm,	Z =   -253.760  mm,
	W =  90.000 deg,	P =   0.000 deg,	R =   90.000 deg
};
P[549]{
   GP1:
	UF : 0, UT : 6,		CONFIG : 'N U T, 0, 0, 0',
	X =  447.604  mm,	Y =   -472.029  mm,	Z =   -254.097  mm,
	W =  90.000 deg,	P =   0.000 deg,	R =   90.000 deg
};
P[550]{
   GP1:
	UF : 0, UT : 6,		CONFIG : 'N U T, 0, 0, 0',
	X =  448.258  mm,	Y =   -471.695  mm,	Z =   -253.991  mm,
	W =  90.000 deg,	P =   0.000 deg,	R =   90.000 deg
};
P[551]{
   GP1:
	UF : 0, UT : 6,		CONFIG : 'N U T, 0, 0, 0',
	X =  449.269  mm,	Y =   -471.151  mm,	Z =   -253.896  mm,
	W =  90.000 deg,	P =   0.000 deg,	R =   90.000 deg
};
P[552]{
   GP1:
	UF : 0, UT : 6,		CONFIG : 'N U T, 0, 0, 0',
	X =  450.076  mm,	Y =   -470.701  mm,	Z =   -253.856  mm,
	W =  90.000 deg,	P =   0.000 deg,	R =   90.000 deg
};
P[553]{
   GP1:
	UF : 0, UT : 6,		CONFIG : 'N U T, 0, 0, 0',
	X =  453.430  mm,	Y =   -468.789  mm,	Z =   -253.797  mm,
	W =  90.000 deg,	P =   0.000 deg,	R =   90.000 deg
};
P[554]{
   GP1:
	UF : 0, UT : 6,		CONFIG : 'N U T, 0, 0, 0',
	X =  454.214  mm,	Y =   -468.248  mm,	Z =   -254.009  mm,
	W =  90.000 deg,	P =   0.000 deg,	R =   90.000 deg
};
P[555]{
   GP1:
	UF : 0, UT : 6,		CONFIG : 'N U T, 0, 0, 0',
	X =  456.354  mm,	Y =   -467.159  mm,	Z =   -253.655  mm,
	W =  90.000 deg,	P =   0.000 deg,	R =   90.000 deg
};
P[556]{
   GP1:
	UF : 0, UT : 6,		CONFIG : 'N U T, 0, 0, 0',
	X =  458.496  mm,	Y =   -465.733  mm,	Z =   -254.115  mm,
	W =  90.000 deg,	P =   0.000 deg,	R =   90.000 deg
};
P[557]{
   GP1:
	UF : 0, UT : 6,		CONFIG : 'N U T, 0, 0, 0',
	X =  460.895  mm,	Y =   -464.481  mm,	Z =   -253.789  mm,
	W =  90.000 deg,	P =   0.000 deg,	R =   90.000 deg
};
P[558]{
   GP1:
	UF : 0, UT : 6,		CONFIG : 'N U T, 0, 0, 0',
	X =  463.396  mm,	Y =   -462.939  mm,	Z =   -254.029  mm,
	W =  90.000 deg,	P =   0.000 deg,	R =   90.000 deg
};
P[559]{
   GP1:
	UF : 0, UT : 6,		CONFIG : 'N U T, 0, 0, 0',
	X =  468.282  mm,	Y =   -460.146  mm,	Z =   -253.959  mm,
	W =  90.000 deg,	P =   0.000 deg,	R =   90.000 deg
};
P[560]{
   GP1:
	UF : 0, UT : 6,		CONFIG : 'N U T, 0, 0, 0',
	X =  471.929  mm,	Y =   -458.020  mm,	Z =   -254.008  mm,
	W =  90.000 deg,	P =   0.000 deg,	R =   90.000 deg
};
P[561]{
   GP1:
	UF : 0, UT : 6,		CONFIG : 'N U T, 0, 0, 0',
	X =  473.387  mm,	Y =   -457.287  mm,	Z =   -253.744  mm,
	W =  90.000 deg,	P =   0.000 deg,	R =   90.000 deg
};
P[562]{
   GP1:
	UF : 0, UT : 6,		CONFIG : 'N U T, 0, 0, 0',
	X =  474.143  mm,	Y =   -456.847  mm,	Z =   -253.753  mm,
	W =  90.000 deg,	P =   0.000 deg,	R =   90.000 deg
};
P[563]{
   GP1:
	UF : 0, UT : 6,		CONFIG : 'N U T, 0, 0, 0',
	X =  475.825  mm,	Y =   -455.752  mm,	Z =   -254.054  mm,
	W =  90.000 deg,	P =   0.000 deg,	R =   90.000 deg
};
P[564]{
   GP1:
	UF : 0, UT : 6,		CONFIG : 'N U T, 0, 0, 0',
	X =  477.142  mm,	Y =   -455.070  mm,	Z =   -253.863  mm,
	W =  90.000 deg,	P =   0.000 deg,	R =   90.000 deg
};
P[565]{
   GP1:
	UF : 0, UT : 6,		CONFIG : 'N U T, 0, 0, 0',
	X =  480.509  mm,	Y =   -453.207  mm,	Z =   -253.669  mm,
	W =  90.000 deg,	P =   0.000 deg,	R =   90.000 deg
};
P[566]{
   GP1:
	UF : 0, UT : 6,		CONFIG : 'N U T, 0, 0, 0',
	X =  484.327  mm,	Y =   -450.964  mm,	Z =   -253.760  mm,
	W =  90.000 deg,	P =   0.000 deg,	R =   90.000 deg
};
P[567]{
   GP1:
	UF : 0, UT : 6,		CONFIG : 'N U T, 0, 0, 0',
	X =  485.317  mm,	Y =   -450.248  mm,	Z =   -254.110  mm,
	W =  90.000 deg,	P =   0.000 deg,	R =   90.000 deg
};
P[568]{
   GP1:
	UF : 0, UT : 6,		CONFIG : 'N U T, 0, 0, 0',
	X =  487.650  mm,	Y =   -449.022  mm,	Z =   -253.818  mm,
	W =  90.000 deg,	P =   0.000 deg,	R =   90.000 deg
};
P[569]{
   GP1:
	UF : 0, UT : 6,		CONFIG : 'N U T, 0, 0, 0',
	X =  489.087  mm,	Y =   -448.167  mm,	Z =   -253.877  mm,
	W =  90.000 deg,	P =   0.000 deg,	R =   90.000 deg
};
P[570]{
   GP1:
	UF : 0, UT : 6,		CONFIG : 'N U T, 0, 0, 0',
	X =  490.367  mm,	Y =   -447.498  mm,	Z =   -253.709  mm,
	W =  90.000 deg,	P =   0.000 deg,	R =   90.000 deg
};
P[571]{
   GP1:
	UF : 0, UT : 6,		CONFIG : 'N U T, 0, 0, 0',
	X =  491.725  mm,	Y =   -446.576  mm,	Z =   -254.041  mm,
	W =  90.000 deg,	P =   0.000 deg,	R =   90.000 deg
};
P[572]{
   GP1:
	UF : 0, UT : 6,		CONFIG : 'N U T, 0, 0, 0',
	X =  494.210  mm,	Y =   -445.184  mm,	Z =   -253.938  mm,
	W =  90.000 deg,	P =   0.000 deg,	R =   90.000 deg
};
P[573]{
   GP1:
	UF : 0, UT : 6,		CONFIG : 'N U T, 0, 0, 0',
	X =  494.942  mm,	Y =   -444.743  mm,	Z =   -253.984  mm,
	W =  90.000 deg,	P =   0.000 deg,	R =   90.000 deg
};
P[574]{
   GP1:
	UF : 0, UT : 6,		CONFIG : 'N U T, 0, 0, 0',
	X =  496.922  mm,	Y =   -443.718  mm,	Z =   -253.698  mm,
	W =  90.000 deg,	P =   0.000 deg,	R =   90.000 deg
};
P[575]{
   GP1:
	UF : 0, UT : 6,		CONFIG : 'N U T, 0, 0, 0',
	X =  498.077  mm,	Y =   -442.946  mm,	Z =   -253.952  mm,
	W =  90.000 deg,	P =   0.000 deg,	R =   90.000 deg
};
P[576]{
   GP1:
	UF : 0, UT : 6,		CONFIG : 'N U T, 0, 0, 0',
	X =  499.757  mm,	Y =   -441.909  mm,	Z =   -254.114  mm,
	W =  90.000 deg,	P =   0.000 deg,	R =   90.000 deg
};
P[577]{
   GP1:
	UF : 0, UT : 6,		CONFIG : 'N U T, 0, 0, 0',
	X =  501.581  mm,	Y =   -440.869  mm,	Z =   -254.083  mm,
	W =  90.000 deg,	P =   0.000 deg,	R =   90.000 deg
};
P[578]{
   GP1:
	UF : 0, UT : 6,		CONFIG : 'N U T, 0, 0, 0',
	X =  503.685  mm,	Y =   -439.834  mm,	Z =   -253.644  mm,
	W =  90.000 deg,	P =   0.000 deg,	R =   90.000 deg
};
P[579]{
   GP1:
	UF : 0, UT : 6,		CONFIG : 'N U T, 0, 0, 0',
	X =  504.486  mm,	Y =   -439.251  mm,	Z =   -253.939  mm,
	W =  90.000 deg,	P =   0.000 deg,	R =   90.000 deg
};
P[580]{
   GP1:
	UF : 0, UT : 6,		CONFIG : 'N U T, 0, 0, 0',
	X =  505.087  mm,	Y =   -438.995  mm,	Z =   -253.718  mm,
	W =  90.000 deg,	P =   0.000 deg,	R =   90.000 deg
};
P[581]{
   GP1:
	UF : 0, UT : 6,		CONFIG : 'N U T, 0, 0, 0',
	X =  506.264  mm,	Y =   -438.153  mm,	Z =   -254.110  mm,
	W =  90.000 deg,	P =   0.000 deg,	R =   90.000 deg
};
P[582]{
   GP1:
	UF : 0, UT : 6,		CONFIG : 'N U T, 0, 0, 0',
	X =  507.449  mm,	Y =   -437.595  mm,	Z =   -253.804  mm,
	W =  90.000 deg,	P =   0.000 deg,	R =   90.000 deg
};
P[583]{
   GP1:
	UF : 0, UT : 6,		CONFIG : 'N U T, 0, 0, 0',
	X =  508.577  mm,	Y =   -436.888  mm,	Z =   -253.942  mm,
	W =  90.000 deg,	P =   0.000 deg,	R =   90.000 deg
};
P[584]{
   GP1:
	UF : 0, UT : 6,		CONFIG : 'N U T, 0, 0, 0',
	X =  511.218  mm,	Y =   -435.287  mm,	Z =   -254.124  mm,
	W =  90.000 deg,	P =   0.000 deg,	R =   90.000 deg
};
P[585]{
   GP1:
	UF : 0, UT : 6,		CONFIG : 'N U T, 0, 0, 0',
	X =  513.918  mm,	Y =   -433.807  mm,	Z =   -253.894  mm,
	W =  90.000 deg,	P =   0.000 deg,	R =   90.000 deg
};
P[586]{
   GP1:
	UF : 0, UT : 6,		CONFIG : 'N U T, 0, 0, 0',
	X =  515.079  mm,	Y =   -433.012  mm,	Z =   -253.792  mm,
	W =  90.000 deg,	P =   0.000 deg,	R =   90.000 deg
};
P[587]{
   GP1:
	UF : 0, UT : 6,		CONFIG : 'N U T, 0, 0, 0',
	X =  517.187  mm,	Y =   -431.094  mm,	Z =   -253.899  mm,
	W =  90.000 deg,	P =   0.000 deg,	R =   90.000 deg
};
P[588]{
   GP1:
	UF : 0, UT : 6,		CONFIG : 'N U T, 0, 0, 0',
	X =  518.793  mm,	Y =   -429.198  mm,	Z =   -253.714  mm,
	W =  90.000 deg,	P =   0.000 deg,	R =   90.000 deg
};
P[589]{
   GP1:
	UF : 0, UT : 6,		CONFIG : 'N U T, 0, 0, 0',
	X =  519.397  mm,	Y =   -427.658  mm,	Z =   -254.116  mm,
	W =  90.000 deg,	P =   0.000 deg,	R =   90.000 deg
};
P[590]{
   GP1:
	UF : 0, UT : 6,		CONFIG : 'N U T, 0, 0, 0',
	X =  520.795  mm,	Y =   -421.542  mm,	Z =   -253.800  mm,
	W =  90.000 deg,	P =   0.000 deg,	R =   90.000 deg
};
P[591]{
   GP1:
	UF : 0, UT : 6,		CONFIG : 'N U T, 0, 0, 0',
	X =  520.618  mm,	Y =   -420.729  mm,	Z =   -254.104  mm,
	W =  90.000 deg,	P =   0.000 deg,	R =   90.000 deg
};
P[592]{
   GP1:
	UF : 0, UT : 6,		CONFIG : 'N U T, 0, 0, 0',
	X =  520.331  mm,	Y =   -419.147  mm,	Z =   -254.037  mm,
	W =  90.000 deg,	P =   0.000 deg,	R =   90.000 deg
};
P[593]{
   GP1:
	UF : 0, UT : 6,		CONFIG : 'N U T, 0, 0, 0',
	X =  519.601  mm,	Y =   -416.463  mm,	Z =   -253.665  mm,
	W =  90.000 deg,	P =   0.000 deg,	R =   90.000 deg
};
P[594]{
   GP1:
	UF : 0, UT : 6,		CONFIG : 'N U T, 0, 0, 0',
	X =  519.014  mm,	Y =   -415.589  mm,	Z =   -254.127  mm,
	W =  90.000 deg,	P =   0.000 deg,	R =   90.000 deg
};
P[595]{
   GP1:
	UF : 0, UT : 6,		CONFIG : 'N U T, 0, 0, 0',
	X =  518.474  mm,	Y =   -414.445  mm,	Z =   -254.028  mm,
	W =  90.000 deg,	P =   0.000 deg,	R =   90.000 deg
};
P[596]{
   GP1:
	UF : 0, UT : 6,		CONFIG : 'N U T, 0, 0, 0',
	X =  517.153  mm,	Y =   -412.036  mm,	Z =   -253.856  mm,
	W =  90.000 deg,	P =   0.000 deg,	R =   90.000 deg
};
P[597]{
   GP1:
	UF : 0, UT : 6,		CONFIG : 'N U T, 0, 0, 0',
	X =  516.678  mm,	Y =   -411.296  mm,	Z =   -253.974  mm,
	W =  90.000 deg,	P =   0.000 deg,	R =   90.000 deg
};
P[598]{
   GP1:
	UF : 0, UT : 6,		CONFIG : 'N U T, 0, 0, 0',
	X =  516.180  mm,	Y =   -410.434  mm,	Z =   -253.973  mm,
	W =  90.000 deg,	P =   0.000 deg,	R =   90.000 deg
};
P[599]{
   GP1:
	UF : 0, UT : 6,		CONFIG : 'N U T, 0, 0, 0',
	X =  515.161  mm,	Y =   -408.709  mm,	Z =   -254.028  mm,
	W =  90.000 deg,	P =   0.000 deg,	R =   90.000 deg
};
P[600]{
   GP1:
	UF : 0, UT : 6,		CONFIG : 'N U T, 0, 0, 0',
	X =  513.798  mm,	Y =   -406.357  mm,	Z =   -254.041  mm,
	W =  90.000 deg,	P =   0.000 deg,	R =   90.000 deg
};
P[601]{
   GP1:
	UF : 0, UT : 6,		CONFIG : 'N U T, 0, 0, 0',
	X =  510.671  mm,	Y =   -400.863  mm,	Z =   -253.934  mm,
	W =  90.000 deg,	P =   0.000 deg,	R =   90.000 deg
};
P[602]{
   GP1:
	UF : 0, UT : 6,		CONFIG : 'N U T, 0, 0, 0',
	X =  509.837  mm,	Y =   -399.318  mm,	Z =   -253.793  mm,
	W =  90.000 deg,	P =   0.000 deg,	R =   90.000 deg
};
P[603]{
   GP1:
	UF : 0, UT : 6,		CONFIG : 'N U T, 0, 0, 0',
	X =  506.775  mm,	Y =   -394.229  mm,	Z =   -254.093  mm,
	W =  90.000 deg,	P =   0.000 deg,	R =   90.000 deg
};
P[604]{
   GP1:
	UF : 0, UT : 6,		CONFIG : 'N U T, 0, 0, 0',
	X =  505.684  mm,	Y =   -392.313  mm,	Z =   -254.053  mm,
	W =  90.000 deg,	P =   0.000 deg,	R =   90.000 deg
};
P[605]{
   GP1:
	UF : 0, UT : 6,		CONFIG : 'N U T, 0, 0, 0',
	X =  503.104  mm,	Y =   -387.751  mm,	Z =   -253.922  mm,
	W =  90.000 deg,	P =   0.000 deg,	R =   90.000 deg
};
P[606]{
   GP1:
	UF : 0, UT : 6,		CONFIG : 'N U T, 0, 0, 0',
	X =  501.763  mm,	Y =   -385.513  mm,	Z =   -254.041  mm,
	W =  90.000 deg,	P =   0.000 deg,	R =   90.000 deg
};
P[607]{
   GP1:
	UF : 0, UT : 6,		CONFIG : 'N U T, 0, 0, 0',
	X =  500.741  mm,	Y =   -383.678  mm,	Z =   -253.948  mm,
	W =  90.000 deg,	P =   0.000 deg,	R =   90.000 deg
};
P[608]{
   GP1:
	UF : 0, UT : 6,		CONFIG : 'N U T, 0, 0, 0',
	X =  500.131  mm,	Y =   -382.559  mm,	Z =   -253.863  mm,
	W =  90.000 deg,	P =   0.000 deg,	R =   90.000 deg
};
P[609]{
   GP1:
	UF : 0, UT : 6,		CONFIG : 'N U T, 0, 0, 0',
	X =  499.318  mm,	Y =   -381.010  mm,	Z =   -253.667  mm,
	W =  90.000 deg,	P =   0.000 deg,	R =   90.000 deg
};
P[610]{
   GP1:
	UF : 0, UT : 6,		CONFIG : 'N U T, 0, 0, 0',
	X =  497.040  mm,	Y =   -377.255  mm,	Z =   -253.933  mm,
	W =  90.000 deg,	P =   0.000 deg,	R =   90.000 deg
};
P[611]{
   GP1:
	UF : 0, UT : 6,		CONFIG : 'N U T, 0, 0, 0',
	X =  495.342  mm,	Y =   -374.425  mm,	Z =   -254.087  mm,
	W =  90.000 deg,	P =   0.000 deg,	R =   90.000 deg
};
P[612]{
   GP1:
	UF : 0, UT : 6,		CONFIG : 'N U T, 0, 0, 0',
	X =  494.988  mm,	Y =   -373.823  mm,	Z =   -254.102  mm,
	W =  90.000 deg,	P =   0.000 deg,	R =   90.000 deg
};
P[613]{
   GP1:
	UF : 0, UT : 6,		CONFIG : 'N U T, 0, 0, 0',
	X =  494.582  mm,	Y =   -372.860  mm,	Z =   -253.739  mm,
	W =  90.000 deg,	P =   0.000 deg,	R =   90.000 deg
};
P[614]{
   GP1:
	UF : 0, UT : 6,		CONFIG : 'N U T, 0, 0, 0',
	X =  493.981  mm,	Y =   -372.084  mm,	Z =   -254.112  mm,
	W =  90.000 deg,	P =   0.000 deg,	R =   90.000 deg
};
P[615]{
   GP1:
	UF : 0, UT : 6,		CONFIG : 'N U T, 0, 0, 0',
	X =  493.085  mm,	Y =   -370.261  mm,	Z =   -253.729  mm,
	W =  90.000 deg,	P =   0.000 deg,	R =   90.000 deg
};
P[616]{
   GP1:
	UF : 0, UT : 6,		CONFIG : 'N U T, 0, 0, 0',
	X =  490.955  mm,	Y =   -366.567  mm,	Z =   -253.725  mm,
	W =  90.000 deg,	P =   0.000 deg,	R =   90.000 deg
};
P[617]{
   GP1:
	UF : 0, UT : 6,		CONFIG : 'N U T, 0, 0, 0',
	X =  490.228  mm,	Y =   -365.577  mm,	Z =   -254.101  mm,
	W =  90.000 deg,	P =   0.000 deg,	R =   90.000 deg
};
P[618]{
   GP1:
	UF : 0, UT : 6,		CONFIG : 'N U T, 0, 0, 0',
	X =  489.724  mm,	Y =   -364.559  mm,	Z =   -253.898  mm,
	W =  90.000 deg,	P =   0.000 deg,	R =   90.000 deg
};
P[619]{
   GP1:
	UF : 0, UT : 6,		CONFIG : 'N U T, 0, 0, 0',
	X =  487.263  mm,	Y =   -360.398  mm,	Z =   -254.037  mm,
	W =  90.000 deg,	P =   0.000 deg,	R =   90.000 deg
};
P[620]{
   GP1:
	UF : 0, UT : 6,		CONFIG : 'N U T, 0, 0, 0',
	X =  486.278  mm,	Y =   -358.679  mm,	Z =   -254.021  mm,
	W =  90.000 deg,	P =   0.000 deg,	R =   90.000 deg
};
P[621]{
   GP1:
	UF : 0, UT : 6,		CONFIG : 'N U T, 0, 0, 0',
	X =  485.348  mm,	Y =   -357.017  mm,	Z =   -253.948  mm,
	W =  90.000 deg,	P =   0.000 deg,	R =   90.000 deg
};
P[622]{
   GP1:
	UF : 0, UT : 6,		CONFIG : 'N U T, 0, 0, 0',
	X =  484.265  mm,	Y =   -355.124  mm,	Z =   -253.924  mm,
	W =  90.000 deg,	P =   0.000 deg,	R =   90.000 deg
};
P[623]{
   GP1:
	UF : 0, UT : 6,		CONFIG : 'N U T, 0, 0, 0',
	X =  483.813  mm,	Y =   -354.449  mm,	Z =   -254.075  mm,
	W =  90.000 deg,	P =   0.000 deg,	R =   90.000 deg
};
P[624]{
   GP1:
	UF : 0, UT : 6,		CONFIG : 'N U T, 0, 0, 0',
	X =  482.216  mm,	Y =   -351.523  mm,	Z =   -253.850  mm,
	W =  90.000 deg,	P =   0.000 deg,	R =   90.000 deg
};
P[625]{
   GP1:
	UF : 0, UT : 6,		CONFIG : 'N U T, 0, 0, 0',
	X =  481.440  mm,	Y =   -350.117  mm,	Z =   -253.766  mm,
	W =  90.000 deg,	P =   0.000 deg,	R =   90.000 deg
};
P[626]{
   GP1:
	UF : 0, UT : 6,		CONFIG : 'N U T, 0, 0, 0',
	X =  479.167  mm,	Y =   -346.356  mm,	Z =   -254.009  mm,
	W =  90.000 deg,	P =   0.000 deg,	R =   90.000 deg
};
P[627]{
   GP1:
	UF : 0, UT : 6,		CONFIG : 'N U T, 0, 0, 0',
	X =  478.621  mm,	Y =   -345.404  mm,	Z =   -254.002  mm,
	W =  90.000 deg,	P =   0.000 deg,	R =   90.000 deg
};
P[628]{
   GP1:
	UF : 0, UT : 6,		CONFIG : 'N U T, 0, 0, 0',
	X =  477.718  mm,	Y =   -343.863  mm,	Z =   -254.034  mm,
	W =  90.000 deg,	P =   0.000 deg,	R =   90.000 deg
};
P[629]{
   GP1:
	UF : 0, UT : 6,		CONFIG : 'N U T, 0, 0, 0',
	X =  476.829  mm,	Y =   -342.293  mm,	Z =   -253.992  mm,
	W =  90.000 deg,	P =   0.000 deg,	R =   90.000 deg
};
P[630]{
   GP1:
	UF : 0, UT : 6,		CONFIG : 'N U T, 0, 0, 0',
	X =  475.555  mm,	Y =   -340.148  mm,	Z =   -254.076  mm,
	W =  90.000 deg,	P =   0.000 deg,	R =   90.000 deg
};
P[631]{
   GP1:
	UF : 0, UT : 6,		CONFIG : 'N U T, 0, 0, 0',
	X =  474.947  mm,	Y =   -339.058  mm,	Z =   -254.026  mm,
	W =  90.000 deg,	P =   0.000 deg,	R =   90.000 deg
};
P[632]{
   GP1:
	UF : 0, UT : 6,		CONFIG : 'N U T, 0, 0, 0',
	X =  474.107  mm,	Y =   -337.421  mm,	Z =   -253.771  mm,
	W =  90.000 deg,	P =   0.000 deg,	R =   90.000 deg
};
P[633]{
   GP1:
	UF : 0, UT : 6,		CONFIG : 'N U T, 0, 0, 0',
	X =  473.364  mm,	Y =   -336.362  mm,	Z =   -254.087  mm,
	W =  90.000 deg,	P =   0.000 deg,	R =   90.000 deg
};
P[634]{
   GP1:
	UF : 0, UT : 6,		CONFIG : 'N U T, 0, 0, 0',
	X =  470.749  mm,	Y =   -331.641  mm,	Z =   -253.821  mm,
	W =  90.000 deg,	P =   0.000 deg,	R =   90.000 deg
};
P[635]{
   GP1:
	UF : 0, UT : 6,		CONFIG : 'N U T, 0, 0, 0',
	X =  469.777  mm,	Y =   -329.898  mm,	Z =   -253.734  mm,
	W =  90.000 deg,	P =   0.000 deg,	R =   90.000 deg
};
P[636]{
   GP1:
	UF : 0, UT : 6,		CONFIG : 'N U T, 0, 0, 0',
	X =  469.311  mm,	Y =   -329.146  mm,	Z =   -253.814  mm,
	W =  90.000 deg,	P =   0.000 deg,	R =   90.000 deg
};
P[637]{
   GP1:
	UF : 0, UT : 6,		CONFIG : 'N U T, 0, 0, 0',
	X =  467.400  mm,	Y =   -325.901  mm,	Z =   -253.906  mm,
	W =  90.000 deg,	P =   0.000 deg,	R =   90.000 deg
};
P[638]{
   GP1:
	UF : 0, UT : 6,		CONFIG : 'N U T, 0, 0, 0',
	X =  466.239  mm,	Y =   -323.928  mm,	Z =   -253.958  mm,
	W =  90.000 deg,	P =   0.000 deg,	R =   90.000 deg
};
P[639]{
   GP1:
	UF : 0, UT : 6,		CONFIG : 'N U T, 0, 0, 0',
	X =  465.846  mm,	Y =   -323.124  mm,	Z =   -253.785  mm,
	W =  90.000 deg,	P =   0.000 deg,	R =   90.000 deg
};
P[640]{
   GP1:
	UF : 0, UT : 6,		CONFIG : 'N U T, 0, 0, 0',
	X =  464.772  mm,	Y =   -321.164  mm,	Z =   -253.644  mm,
	W =  90.000 deg,	P =   0.000 deg,	R =   90.000 deg
};
P[641]{
   GP1:
	UF : 0, UT : 6,		CONFIG : 'N U T, 0, 0, 0',
	X =  463.014  mm,	Y =   -318.129  mm,	Z =   -253.658  mm,
	W =  90.000 deg,	P =   0.000 deg,	R =   90.000 deg
};
P[642]{
   GP1:
	UF : 0, UT : 6,		CONFIG : 'N U T, 0, 0, 0',
	X =  462.350  mm,	Y =   -317.082  mm,	Z =   -253.802  mm,
	W =  90.000 deg,	P =   0.000 deg,	R =   90.000 deg
};
P[643]{
   GP1:
	UF : 0, UT : 6,		CONFIG : 'N U T, 0, 0, 0',
	X =  460.789  mm,	Y =   -314.509  mm,	Z =   -253.984  mm,
	W =  90.000 deg,	P =   0.000 deg,	R =   90.000 deg
};
P[644]{
   GP1:
	UF : 0, UT : 6,		CONFIG : 'N U T, 0, 0, 0',
	X =  460.507  mm,	Y =   -313.888  mm,	Z =   -253.802  mm,
	W =  90.000 deg,	P =   0.000 deg,	R =   90.000 deg
};
P[645]{
   GP1:
	UF : 0, UT : 6,		CONFIG : 'N U T, 0, 0, 0',
	X =  459.032  mm,	Y =   -311.298  mm,	Z =   -253.750  mm,
	W =  90.000 deg,	P =   0.000 deg,	R =   90.000 deg
};
P[646]{
   GP1:
	UF : 0, UT : 6,		CONFIG : 'N U T, 0, 0, 0',
	X =  458.214  mm,	Y =   -309.904  mm,	Z =   -253.782  mm,
	W =  90.000 deg,	P =   0.000 deg,	R =   90.000 deg
};
P[647]{
   GP1:
	UF : 0, UT : 6,		CONFIG : 'N U T, 0, 0, 0',
	X =  457.392  mm,	Y =   -308.696  mm,	Z =   -254.084  mm,
	W =  90.000 deg,	P =   0.000 deg,	R =   90.000 deg
};
P[648]{
   GP1:
	UF : 0, UT : 6,		CONFIG : 'N U T, 0, 0, 0',
	X =  456.349  mm,	Y =   -306.874  mm,	Z =   -254.063  mm,
	W =  90.000 deg,	P =   0.000 deg,	R =   90.000 deg
};
P[649]{
   GP1:
	UF : 0, UT : 6,		CONFIG : 'N U T, 0, 0, 0',
	X =  455.204  mm,	Y =   -304.638  mm,	Z =   -253.708  mm,
	W =  90.000 deg,	P =   0.000 deg,	R =   90.000 deg
};
P[650]{
   GP1:
	UF : 0, UT : 6,		CONFIG : 'N U T, 0, 0, 0',
	X =  454.659  mm,	Y =   -303.713  mm,	Z =   -253.736  mm,
	W =  90.000 deg,	P =   0.000 deg,	R =   90.000 deg
};
P[651]{
   GP1:
	UF : 0, UT : 6,		CONFIG : 'N U T, 0, 0, 0',
	X =  454.262  mm,	Y =   -303.120  mm,	Z =   -253.866  mm,
	W =  90.000 deg,	P =   0.000 deg,	R =   90.000 deg
};
P[652]{
   GP1:
	UF : 0, UT : 6,		CONFIG : 'N U T, 0, 0, 0',
	X =  451.217  mm,	Y =   -297.902  mm,	Z =   -253.945  mm,
	W =  90.000 deg,	P =   0.000 deg,	R =   90.000 deg
};
P[653]{
   GP1:
	UF : 0, UT : 6,		CONFIG : 'N U T, 0, 0, 0',
	X =  450.663  mm,	Y =   -296.793  mm,	Z =   -253.735  mm,
	W =  90.000 deg,	P =   0.000 deg,	R =   90.000 deg
};
P[654]{
   GP1:
	UF : 0, UT : 6,		CONFIG : 'N U T, 0, 0, 0',
	X =  448.117  mm,	Y =   -292.519  mm,	Z =   -253.924  mm,
	W =  90.000 deg,	P =   0.000 deg,	R =   90.000 deg
};
P[655]{
   GP1:
	UF : 0, UT : 6,		CONFIG : 'N U T, 0, 0, 0',
	X =  447.132  mm,	Y =   -290.933  mm,	Z =   -254.092  mm,
	W =  90.000 deg,	P =   0.000 deg,	R =   90.000 deg
};
P[656]{
   GP1:
	UF : 0, UT : 6,		CONFIG : 'N U T, 0, 0, 0',
	X =  446.824  mm,	Y =   -290.112  mm,	Z =   -253.690  mm,
	W =  90.000 deg,	P =   0.000 deg,	R =   90.000 deg
};
P[657]{
   GP1:
	UF : 0, UT : 6,		CONFIG : 'N U T, 0, 0, 0',
	X =  446.022  mm,	Y =   -288.795  mm,	Z =   -253.792  mm,
	W =  90.000 deg,	P =   0.000 deg,	R =   90.000 deg
};
P[658]{
   GP1:
	UF : 0, UT : 6,		CONFIG : 'N U T, 0, 0, 0',
	X =  444.935  mm,	Y =   -287.109  mm,	Z =   -254.068  mm,
	W =  90.000 deg,	P =   0.000 deg,	R =   90.000 deg
};
P[659]{
   GP1:
	UF : 0, UT : 6,		CONFIG : 'N U T, 0, 0, 0',
	X =  444.095  mm,	Y =   -285.488  mm,	Z =   -253.835  mm,
	W =  90.000 deg,	P =   0.000 deg,	R =   90.000 deg
};
P[660]{
   GP1:
	UF : 0, UT : 6,		CONFIG : 'N U T, 0, 0, 0',
	X =  442.092  mm,	Y =   -281.997  mm,	Z =   -253.805  mm,
	W =  90.000 deg,	P =   0.000 deg,	R =   90.000 deg
};
P[661]{
   GP1:
	UF : 0, UT : 6,		CONFIG : 'N U T, 0, 0, 0',
	X =  441.169  mm,	Y =   -280.318  mm,	Z =   -253.691  mm,
	W =  90.000 deg,	P =   0.000 deg,	R =   90.000 deg
};
P[662]{
   GP1:
	UF : 0, UT : 6,		CONFIG : 'N U T, 0, 0, 0',
	X =  440.819  mm,	Y =   -279.667  mm,	Z =   -253.629  mm,
	W =  90.000 deg,	P =   0.000 deg,	R =   90.000 deg
};
P[663]{
   GP1:
	UF : 0, UT : 6,		CONFIG : 'N U T, 0, 0, 0',
	X =  439.379  mm,	Y =   -277.302  mm,	Z =   -253.807  mm,
	W =  90.000 deg,	P =   0.000 deg,	R =   90.000 deg
};
P[664]{
   GP1:
	UF : 0, UT : 6,		CONFIG : 'N U T, 0, 0, 0',
	X =  438.481  mm,	Y =   -275.884  mm,	Z =   -254.002  mm,
	W =  90.000 deg,	P =   0.000 deg,	R =   90.000 deg
};
P[665]{
   GP1:
	UF : 0, UT : 6,		CONFIG : 'N U T, 0, 0, 0',
	X =  438.117  mm,	Y =   -275.000  mm,	Z =   -253.645  mm,
	W =  90.000 deg,	P =   0.000 deg,	R =   90.000 deg
};
P[666]{
   GP1:
	UF : 0, UT : 6,		CONFIG : 'N U T, 0, 0, 0',
	X =  435.727  mm,	Y =   -271.161  mm,	Z =   -254.068  mm,
	W =  90.000 deg,	P =   0.000 deg,	R =   90.000 deg
};
P[667]{
   GP1:
	UF : 0, UT : 6,		CONFIG : 'N U T, 0, 0, 0',
	X =  435.257  mm,	Y =   -270.219  mm,	Z =   -253.885  mm,
	W =  90.000 deg,	P =   0.000 deg,	R =   90.000 deg
};
P[668]{
   GP1:
	UF : 0, UT : 6,		CONFIG : 'N U T, 0, 0, 0',
	X =  434.689  mm,	Y =   -269.172  mm,	Z =   -253.800  mm,
	W =  90.000 deg,	P =   0.000 deg,	R =   90.000 deg
};
P[669]{
   GP1:
	UF : 0, UT : 6,		CONFIG : 'N U T, 0, 0, 0',
	X =  433.922  mm,	Y =   -267.979  mm,	Z =   -253.988  mm,
	W =  90.000 deg,	P =   0.000 deg,	R =   90.000 deg
};
P[670]{
   GP1:
	UF : 0, UT : 6,		CONFIG : 'N U T, 0, 0, 0',
	X =  432.453  mm,	Y =   -265.269  mm,	Z =   -253.755  mm,
	W =  90.000 deg,	P =   0.000 deg,	R =   90.000 deg
};
P[671]{
   GP1:
	UF : 0, UT : 6,		CONFIG : 'N U T, 0, 0, 0',
	X =  432.030  mm,	Y =   -264.797  mm,	Z =   -254.121  mm,
	W =  90.000 deg,	P =   0.000 deg,	R =   90.000 deg
};
P[672]{
   GP1:
	UF : 0, UT : 6,		CONFIG : 'N U T, 0, 0, 0',
	X =  431.508  mm,	Y =   -263.882  mm,	Z =   -254.105  mm,
	W =  90.000 deg,	P =   0.000 deg,	R =   90.000 deg
};
P[673]{
   GP1:
	UF : 0, UT : 6,		CONFIG : 'N U T, 0, 0, 0',
	X =  431.008  mm,	Y =   -262.759  mm,	Z =   -253.747  mm,
	W =  90.000 deg,	P =   0.000 deg,	R =   90.000 deg
};
P[674]{
   GP1:
	UF : 0, UT : 6,		CONFIG : 'N U T, 0, 0, 0',
	X =  430.324  mm,	Y =   -261.658  mm,	Z =   -253.860  mm,
	W =  90.000 deg,	P =   0.000 deg,	R =   90.000 deg
};
P[675]{
   GP1:
	UF : 0, UT : 6,		CONFIG : 'N U T, 0, 0, 0',
	X =  429.688  mm,	Y =   -260.558  mm,	Z =   -253.865  mm,
	W =  90.000 deg,	P =   0.000 deg,	R =   90.000 deg
};
P[676]{
   GP1:
	UF : 0, UT : 6,		CONFIG : 'N U T, 0, 0, 0',
	X =  427.571  mm,	Y =   -256.807  mm,	Z =   -253.747  mm,
	W =  90.000 deg,	P =   0.000 deg,	R =   90.000 deg
};
P[677]{
   GP1:
	UF : 0, UT : 6,		CONFIG : 'N U T, 0, 0, 0',
	X =  425.846  mm,	Y =   -253.958  mm,	Z =   -253.942  mm,
	W =  90.000 deg,	P =   0.000 deg,	R =   90.000 deg
};
P[678]{
   GP1:
	UF : 0, UT : 6,		CONFIG : 'N U T, 0, 0, 0',
	X =  425.450  mm,	Y =   -253.170  mm,	Z =   -253.796  mm,
	W =  90.000 deg,	P =   0.000 deg,	R =   90.000 deg
};
P[679]{
   GP1:
	UF : 0, UT : 6,		CONFIG : 'N U T, 0, 0, 0',
	X =  423.883  mm,	Y =   -250.445  mm,	Z =   -253.782  mm,
	W =  90.000 deg,	P =   0.000 deg,	R =   90.000 deg
};
P[680]{
   GP1:
	UF : 0, UT : 6,		CONFIG : 'N U T, 0, 0, 0',
	X =  422.722  mm,	Y =   -248.633  mm,	Z =   -254.059  mm,
	W =  90.000 deg,	P =   0.000 deg,	R =   90.000 deg
};
P[681]{
   GP1:
	UF : 0, UT : 6,		CONFIG : 'N U T, 0, 0, 0',
	X =  421.935  mm,	Y =   -246.981  mm,	Z =   -253.656  mm,
	W =  90.000 deg,	P =   0.000 deg,	R =   90.000 deg
};
P[682]{
   GP1:
	UF : 0, UT : 6,		CONFIG : 'N U T, 0, 0, 0',
	X =  421.444  mm,	Y =   -246.314  mm,	Z =   -253.912  mm,
	W =  90.000 deg,	P =   0.000 deg,	R =   90.000 deg
};
P[683]{
   GP1:
	UF : 0, UT : 6,		CONFIG : 'N U T, 0, 0, 0',
	X =  420.384  mm,	Y =   -244.600  mm,	Z =   -254.084  mm,
	W =  90.000 deg,	P =   0.000 deg,	R =   90.000 deg
};
P[684]{
   GP1:
	UF : 0, UT : 6,		CONFIG : 'N U T, 0, 0, 0',
	X =  418.104  mm,	Y =   -240.360  mm,	Z =   -253.675  mm,
	W =  90.000 deg,	P =   0.000 deg,	R =   90.000 deg
};
P[685]{
   GP1:
	UF : 0, UT : 6,		CONFIG : 'N U T, 0, 0, 0',
	X =  417.242  mm,	Y =   -239.069  mm,	Z =   -253.957  mm,
	W =  90.000 deg,	P =   0.000 deg,	R =   90.000 deg
};
P[686]{
   GP1:
	UF : 0, UT : 6,		CONFIG : 'N U T, 0, 0, 0',
	X =  416.282  mm,	Y =   -237.349  mm,	Z =   -253.878  mm,
	W =  90.000 deg,	P =   0.000 deg,	R =   90.000 deg
};
P[687]{
   GP1:
	UF : 0, UT : 6,		CONFIG : 'N U T, 0, 0, 0',
	X =  415.254  mm,	Y =   -235.507  mm,	Z =   -253.789  mm,
	W =  90.000 deg,	P =   0.000 deg,	R =   90.000 deg
};
P[688]{
   GP1:
	UF : 0, UT : 6,		CONFIG : 'N U T, 0, 0, 0',
	X =  414.341  mm,	Y =   -233.952  mm,	Z =   -253.829  mm,
	W =  90.000 deg,	P =   0.000 deg,	R =   90.000 deg
};
P[689]{
   GP1:
	UF : 0, UT : 6,		CONFIG : 'N U T, 0, 0, 0',
	X =  411.104  mm,	Y =   -228.309  mm,	Z =   -253.777  mm,
	W =  90.000 deg,	P =   0.000 deg,	R =   90.000 deg
};
P[690]{
   GP1:
	UF : 0, UT : 6,		CONFIG : 'N U T, 0, 0, 0',
	X =  408.913  mm,	Y =   -224.422  mm,	Z =   -253.648  mm,
	W =  90.000 deg,	P =   0.000 deg,	R =   90.000 deg
};
P[691]{
   GP1:
	UF : 0, UT : 6,		CONFIG : 'N U T, 0, 0, 0',
	X =  407.503  mm,	Y =   -222.244  mm,	Z =   -254.018  mm,
	W =  90.000 deg,	P =   0.000 deg,	R =   90.000 deg
};
P[692]{
   GP1:
	UF : 0, UT : 6,		CONFIG : 'N U T, 0, 0, 0',
	X =  406.402  mm,	Y =   -220.079  mm,	Z =   -253.656  mm,
	W =  90.000 deg,	P =   0.000 deg,	R =   90.000 deg
};
P[693]{
   GP1:
	UF : 0, UT : 6,		CONFIG : 'N U T, 0, 0, 0',
	X =  405.344  mm,	Y =   -218.238  mm,	Z =   -253.644  mm,
	W =  90.000 deg,	P =   0.000 deg,	R =   90.000 deg
};
P[694]{
   GP1:
	UF : 0, UT : 6,		CONFIG : 'N U T, 0, 0, 0',
	X =  404.102  mm,	Y =   -216.178  mm,	Z =   -253.769  mm,
	W =  90.000 deg,	P =   0.000 deg,	R =   90.000 deg
};
P[695]{
   GP1:
	UF : 0, UT : 6,		CONFIG : 'N U T, 0, 0, 0',
	X =  403.309  mm,	Y =   -214.834  mm,	Z =   -253.811  mm,
	W =  90.000 deg,	P =   0.000 deg,	R =   90.000 deg
};
P[696]{
   GP1:
	UF : 0, UT : 6,		CONFIG : 'N U T, 0, 0, 0',
	X =  402.814  mm,	Y =   -214.063  mm,	Z =   -253.932  mm,
	W =  90.000 deg,	P =   0.000 deg,	R =   90.000 deg
};
P[697]{
   GP1:
	UF : 0, UT : 6,		CONFIG : 'N U T, 0, 0, 0',
	X =  402.335  mm,	Y =   -213.194  mm,	Z =   -253.877  mm,
	W =  90.000 deg,	P =   0.000 deg,	R =   90.000 deg
};
P[698]{
   GP1:
	UF : 0, UT : 6,		CONFIG : 'N U T, 0, 0, 0',
	X =  401.673  mm,	Y =   -212.073  mm,	Z =   -253.914  mm,
	W =  90.000 deg,	P =   0.000 deg,	R =   90.000 deg
};
P[699]{
   GP1:
	UF : 0, UT : 6,		CONFIG : 'N U T, 0, 0, 0',
	X =  399.212  mm,	Y =   -207.863  mm,	Z =   -253.989  mm,
	W =  90.000 deg,	P =   0.000 deg,	R =   90.000 deg
};
P[700]{
   GP1:
	UF : 0, UT : 6,		CONFIG : 'N U T, 0, 0, 0',
	X =  398.721  mm,	Y =   -206.786  mm,	Z =   -253.670  mm,
	W =  90.000 deg,	P =   0.000 deg,	R =   90.000 deg
};
P[701]{
   GP1:
	UF : 0, UT : 6,		CONFIG : 'N U T, 0, 0, 0',
	X =  397.041  mm,	Y =   -204.180  mm,	Z =   -254.095  mm,
	W =  90.000 deg,	P =   0.000 deg,	R =   90.000 deg
};
P[702]{
   GP1:
	UF : 0, UT : 6,		CONFIG : 'N U T, 0, 0, 0',
	X =  395.008  mm,	Y =   -200.551  mm,	Z =   -253.943  mm,
	W =  90.000 deg,	P =   0.000 deg,	R =   90.000 deg
};
P[703]{
   GP1:
	UF : 0, UT : 6,		CONFIG : 'N U T, 0, 0, 0',
	X =  393.992  mm,	Y =   -198.864  mm,	Z =   -254.045  mm,
	W =  90.000 deg,	P =   0.000 deg,	R =   90.000 deg
};
P[704]{
   GP1:
	UF : 0, UT : 6,		CONFIG : 'N U T, 0, 0, 0',
	X =  392.307  mm,	Y =   -195.782  mm,	Z =   -253.813  mm,
	W =  90.000 deg,	P =   0.000 deg,	R =   90.000 deg
};
P[705]{
   GP1:
	UF : 0, UT : 6,		CONFIG : 'N U T, 0, 0, 0',
	X =  391.914  mm,	Y =   -195.139  mm,	Z =   -253.869  mm,
	W =  90.000 deg,	P =   0.000 deg,	R =   90.000 deg
};
P[706]{
   GP1:
	UF : 0, UT : 6,		CONFIG : 'N U T, 0, 0, 0',
	X =  389.574  mm,	Y =   -190.947  mm,	Z =   -253.673  mm,
	W =  90.000 deg,	P =   0.000 deg,	R =   90.000 deg
};
P[707]{
   GP1:
	UF : 0, UT : 6,		CONFIG : 'N U T, 0, 0, 0',
	X =  388.995  mm,	Y =   -190.188  mm,	Z =   -254.014  mm,
	W =  90.000 deg,	P =   0.000 deg,	R =   90.000 deg
};
P[708]{
   GP1:
	UF : 0, UT : 6,		CONFIG : 'N U T, 0, 0, 0',
	X =  384.284  mm,	Y =   -181.868  mm,	Z =   -253.789  mm,
	W =  90.000 deg,	P =   0.000 deg,	R =   90.000 deg
};
P[709]{
   GP1:
	UF : 0, UT : 6,		CONFIG : 'N U T, 0, 0, 0',
	X =  383.430  mm,	Y =   -180.489  mm,	Z =   -253.932  mm,
	W =  90.000 deg,	P =   0.000 deg,	R =   90.000 deg
};
P[710]{
   GP1:
	UF : 0, UT : 6,		CONFIG : 'N U T, 0, 0, 0',
	X =  382.686  mm,	Y =   -179.043  mm,	Z =   -253.709  mm,
	W =  90.000 deg,	P =   0.000 deg,	R =   90.000 deg
};
P[711]{
   GP1:
	UF : 0, UT : 6,		CONFIG : 'N U T, 0, 0, 0',
	X =  382.247  mm,	Y =   -178.313  mm,	Z =   -253.753  mm,
	W =  90.000 deg,	P =   0.000 deg,	R =   90.000 deg
};
P[712]{
   GP1:
	UF : 0, UT : 6,		CONFIG : 'N U T, 0, 0, 0',
	X =  381.699  mm,	Y =   -177.450  mm,	Z =   -253.872  mm,
	W =  90.000 deg,	P =   0.000 deg,	R =   90.000 deg
};
P[713]{
   GP1:
	UF : 0, UT : 6,		CONFIG : 'N U T, 0, 0, 0',
	X =  380.105  mm,	Y =   -174.665  mm,	Z =   -253.838  mm,
	W =  90.000 deg,	P =   0.000 deg,	R =   90.000 deg
};
P[714]{
   GP1:
	UF : 0, UT : 6,		CONFIG : 'N U T, 0, 0, 0',
	X =  376.046  mm,	Y =   -167.767  mm,	Z =   -254.023  mm,
	W =  90.000 deg,	P =   0.000 deg,	R =   90.000 deg
};
P[715]{
   GP1:
	UF : 0, UT : 6,		CONFIG : 'N U T, 0, 0, 0',
	X =  375.552  mm,	Y =   -166.899  mm,	Z =   -254.006  mm,
	W =  90.000 deg,	P =   0.000 deg,	R =   90.000 deg
};
P[716]{
   GP1:
	UF : 0, UT : 6,		CONFIG : 'N U T, 0, 0, 0',
	X =  375.127  mm,	Y =   -166.236  mm,	Z =   -254.109  mm,
	W =  90.000 deg,	P =   0.000 deg,	R =   90.000 deg
};
P[717]{
   GP1:
	UF : 0, UT : 6,		CONFIG : 'N U T, 0, 0, 0',
	X =  373.896  mm,	Y =   -163.762  mm,	Z =   -253.629  mm,
	W =  90.000 deg,	P =   0.000 deg,	R =   90.000 deg
};
P[718]{
   GP1:
	UF : 0, UT : 6,		CONFIG : 'N U T, 0, 0, 0',
	X =  373.270  mm,	Y =   -162.989  mm,	Z =   -254.065  mm,
	W =  90.000 deg,	P =   0.000 deg,	R =   90.000 deg
};
P[719]{
   GP1:
	UF : 0, UT : 6,		CONFIG : 'N U T, 0, 0, 0',
	X =  372.447  mm,	Y =   -161.370  mm,	Z =   -253.793  mm,
	W =  90.000 deg,	P =   0.000 deg,	R =   90.000 deg
};
P[720]{
   GP1:
	UF : 0, UT : 6,		CONFIG : 'N U T, 0, 0, 0',
	X =  370.541  mm,	Y =   -158.065  mm,	Z =   -253.789  mm,
	W =  90.000 deg,	P =   0.000 deg,	R =   90.000 deg
};
P[721]{
   GP1:
	UF : 0, UT : 6,		CONFIG : 'N U T, 0, 0, 0',
	X =  369.320  mm,	Y =   -155.938  mm,	Z =   -253.770  mm,
	W =  90.000 deg,	P =   0.000 deg,	R =   90.000 deg
};
P[722]{
   GP1:
	UF : 0, UT : 6,		CONFIG : 'N U T, 0, 0, 0',
	X =  368.003  mm,	Y =   -153.771  mm,	Z =   -253.929  mm,
	W =  90.000 deg,	P =   0.000 deg,	R =   90.000 deg
};
P[723]{
   GP1:
	UF : 0, UT : 6,		CONFIG : 'N U T, 0, 0, 0',
	X =  367.685  mm,	Y =   -153.038  mm,	Z =   -253.673  mm,
	W =  90.000 deg,	P =   0.000 deg,	R =   90.000 deg
};
P[724]{
   GP1:
	UF : 0, UT : 6,		CONFIG : 'N U T, 0, 0, 0',
	X =  365.864  mm,	Y =   -150.107  mm,	Z =   -253.989  mm,
	W =  90.000 deg,	P =   0.000 deg,	R =   90.000 deg
};
P[725]{
   GP1:
	UF : 0, UT : 6,		CONFIG : 'N U T, 0, 0, 0',
	X =  365.451  mm,	Y =   -149.220  mm,	Z =   -253.746  mm,
	W =  90.000 deg,	P =   0.000 deg,	R =   90.000 deg
};
P[726]{
   GP1:
	UF : 0, UT : 6,		CONFIG : 'N U T, 0, 0, 0',
	X =  363.625  mm,	Y =   -145.993  mm,	Z =   -253.656  mm,
	W =  90.000 deg,	P =   0.000 deg,	R =   90.000 deg
};
P[727]{
   GP1:
	UF : 0, UT : 6,		CONFIG : 'N U T, 0, 0, 0',
	X =  363.140  mm,	Y =   -145.254  mm,	Z =   -253.798  mm,
	W =  90.000 deg,	P =   0.000 deg,	R =   90.000 deg
};
P[728]{
   GP1:
	UF : 0, UT : 6,		CONFIG : 'N U T, 0, 0, 0',
	X =  362.742  mm,	Y =   -144.750  mm,	Z =   -254.056  mm,
	W =  90.000 deg,	P =   0.000 deg,	R =   90.000 deg
};
P[729]{
   GP1:
	UF : 0, UT : 6,		CONFIG : 'N U T, 0, 0, 0',
	X =  362.154  mm,	Y =   -143.485  mm,	Z =   -253.712  mm,
	W =  90.000 deg,	P =   0.000 deg,	R =   90.000 deg
};
P[730]{
   GP1:
	UF : 0, UT : 6,		CONFIG : 'N U T, 0, 0, 0',
	X =  361.140  mm,	Y =   -141.840  mm,	Z =   -253.867  mm,
	W =  90.000 deg,	P =   0.000 deg,	R =   90.000 deg
};
P[731]{
   GP1:
	UF : 0, UT : 6,		CONFIG : 'N U T, 0, 0, 0',
	X =  360.706  mm,	Y =   -141.009  mm,	Z =   -253.758  mm,
	W =  90.000 deg,	P =   0.000 deg,	R =   90.000 deg
};
P[732]{
   GP1:
	UF : 0, UT : 6,		CONFIG : 'N U T, 0, 0, 0',
	X =  359.670  mm,	Y =   -139.136  mm,	Z =   -253.643  mm,
	W =  90.000 deg,	P =   0.000 deg,	R =   90.000 deg
};
P[733]{
   GP1:
	UF : 0, UT : 6,		CONFIG : 'N U T, 0, 0, 0',
	X =  358.604  mm,	Y =   -137.532  mm,	Z =   -253.987  mm,
	W =  90.000 deg,	P =   0.000 deg,	R =   90.000 deg
};
P[734]{
   GP1:
	UF : 0, UT : 6,		CONFIG : 'N U T, 0, 0, 0',
	X =  357.547  mm,	Y =   -135.637  mm,	Z =   -253.894  mm,
	W =  90.000 deg,	P =   0.000 deg,	R =   90.000 deg
};
P[735]{
   GP1:
	UF : 0, UT : 6,		CONFIG : 'N U T, 0, 0, 0',
	X =  356.528  mm,	Y =   -133.928  mm,	Z =   -253.974  mm,
	W =  90.000 deg,	P =   0.000 deg,	R =   90.000 deg
};
P[736]{
   GP1:
	UF : 0, UT : 6,		CONFIG : 'N U T, 0, 0, 0',
	X =  355.181  mm,	Y =   -131.513  mm,	Z =   -253.859  mm,
	W =  90.000 deg,	P =   0.000 deg,	R =   90.000 deg
};
P[737]{
   GP1:
	UF : 0, UT : 6,		CONFIG : 'N U T, 0, 0, 0',
	X =  354.688  mm,	Y =   -130.669  mm,	Z =   -253.874  mm,
	W =  90.000 deg,	P =   0.000 deg,	R =   90.000 deg
};
P[738]{
   GP1:
	UF : 0, UT : 6,		CONFIG : 'N U T, 0, 0, 0',
	X =  353.472  mm,	Y =   -128.638  mm,	Z =   -253.976  mm,
	W =  90.000 deg,	P =   0.000 deg,	R =   90.000 deg
};
P[739]{
   GP1:
	UF : 0, UT : 6,		CONFIG : 'N U T, 0, 0, 0',
	X =  352.833  mm,	Y =   -127.321  mm,	Z =   -253.684  mm,
	W =  90.000 deg,	P =   0.000 deg,	R =   90.000 deg
};
P[740]{
   GP1:
	UF : 0, UT : 6,		CONFIG : 'N U T, 0, 0, 0',
	X =  351.635  mm,	Y =   -125.831  mm,	Z =   -254.046  mm,
	W =  90.000 deg,	P =   0.000 deg,	R =   90.000 deg
};
P[741]{
   GP1:
	UF : 0, UT : 6,		CONFIG : 'N U T, 0, 0, 0',
	X =  350.971  mm,	Y =   -124.965  mm,	Z =   -254.114  mm,
	W =  90.000 deg,	P =   0.000 deg,	R =   90.000 deg
};
P[742]{
   GP1:
	UF : 0, UT : 6,		CONFIG : 'N U T, 0, 0, 0',
	X =  350.418  mm,	Y =   -124.216  mm,	Z =   -253.920  mm,
	W =  90.000 deg,	P =   0.000 deg,	R =   90.000 deg
};
P[743]{
   GP1:
	UF : 0, UT : 6,		CONFIG : 'N U T, 0, 0, 0',
	X =  345.027  mm,	Y =   -120.731  mm,	Z =   -253.842  mm,
	W =  90.000 deg,	P =   0.000 deg,	R =   90.000 deg
};
P[744]{
   GP1:
	UF : 0, UT : 6,		CONFIG : 'N U T, 0, 0, 0',
	X =  343.176  mm,	Y =   -120.265  mm,	Z =   -253.900  mm,
	W =  90.000 deg,	P =   0.000 deg,	R =   90.000 deg
};
P[745]{
   GP1:
	UF : 0, UT : 6,		CONFIG : 'N U T, 0, 0, 0',
	X =  340.081  mm,	Y =   -120.136  mm,	Z =   -254.039  mm,
	W =  90.000 deg,	P =   0.000 deg,	R =   90.000 deg
};
P[746]{
   GP1:
	UF : 0, UT : 6,		CONFIG : 'N U T, 0, 0, 0',
	X =  338.075  mm,	Y =   -120.414  mm,	Z =   -253.994  mm,
	W =  90.000 deg,	P =   0.000 deg,	R =   90.000 deg
};
P[747]{
   GP1:
	UF : 0, UT : 6,		CONFIG : 'N U T, 0, 0, 0',
	X =  337.128  mm,	Y =   -120.556  mm,	Z =   -253.891  mm,
	W =  90.000 deg,	P =   0.000 deg,	R =   90.000 deg
};
P[748]{
   GP1:
	UF : 0, UT : 6,		CONFIG : 'N U T, 0, 0, 0',
	X =  336.175  mm,	Y =   -120.853  mm,	Z =   -253.896  mm,
	W =  90.000 deg,	P =   0.000 deg,	R =   90.000 deg
};
P[749]{
   GP1:
	UF : 0, UT : 6,		CONFIG : 'N U T, 0, 0, 0',
	X =  335.098  mm,	Y =   -121.407  mm,	Z =   -254.072  mm,
	W =  90.000 deg,	P =   0.000 deg,	R =   90.000 deg
};
P[750]{
   GP1:
	UF : 0, UT : 6,		CONFIG : 'N U T, 0, 0, 0',
	X =  333.932  mm,	Y =   -121.946  mm,	Z =   -254.122  mm,
	W =  90.000 deg,	P =   0.000 deg,	R =   90.000 deg
};
P[751]{
   GP1:
	UF : 0, UT : 6,		CONFIG : 'N U T, 0, 0, 0',
	X =  332.616  mm,	Y =   -122.663  mm,	Z =   -254.099  mm,
	W =  90.000 deg,	P =   0.000 deg,	R =   90.000 deg
};
P[752]{
   GP1:
	UF : 0, UT : 6,		CONFIG : 'N U T, 0, 0, 0',
	X =  332.007  mm,	Y =   -122.919  mm,	Z =   -253.869  mm,
	W =  90.000 deg,	P =   0.000 deg,	R =   90.000 deg
};
P[753]{
   GP1:
	UF : 0, UT : 6,		CONFIG : 'N U T, 0, 0, 0',
	X =  330.502  mm,	Y =   -123.821  mm,	Z =   -253.949  mm,
	W =  90.000 deg,	P =   0.000 deg,	R =   90.000 deg
};
P[754]{
   GP1:
	UF : 0, UT : 6,		CONFIG : 'N U T, 0, 0, 0',
	X =  329.404  mm,	Y =   -124.529  mm,	Z =   -254.128  mm,
	W =  90.000 deg,	P =   0.000 deg,	R =   90.000 deg
};
P[755]{
   GP1:
	UF : 0, UT : 6,		CONFIG : 'N U T, 0, 0, 0',
	X =  328.297  mm,	Y =   -125.029  mm,	Z =   -253.791  mm,
	W =  90.000 deg,	P =   0.000 deg,	R =   90.000 deg
};
P[756]{
   GP1:
	UF : 0, UT : 6,		CONFIG : 'N U T, 0, 0, 0',
	X =  326.612  mm,	Y =   -126.005  mm,	Z =   -253.799  mm,
	W =  90.000 deg,	P =   0.000 deg,	R =   90.000 deg
};
P[757]{
   GP1:
	UF : 0, UT : 6,		CONFIG : 'N U T, 0, 0, 0',
	X =  324.699  mm,	Y =   -127.110  mm,	Z =   -253.799  mm,
	W =  90.000 deg,	P =   0.000 deg,	R =   90.000 deg
};
P[758]{
   GP1:
	UF : 0, UT : 6,		CONFIG : 'N U T, 0, 0, 0',
	X =  324.045  mm,	Y =   -127.614  mm,	Z =   -254.105  mm,
	W =  90.000 deg,	P =   0.000 deg,	R =   90.000 deg
};
P[759]{
   GP1:
	UF : 0, UT : 6,		CONFIG : 'N U T, 0, 0, 0',
	X =  323.292  mm,	Y =   -127.920  mm,	Z =   -253.794  mm,
	W =  90.000 deg,	P =   0.000 deg,	R =   90.000 deg
};
P[760]{
   GP1:
	UF : 0, UT : 6,		CONFIG : 'N U T, 0, 0, 0',
	X =  322.564  mm,	Y =   -128.293  mm,	Z =   -253.677  mm,
	W =  90.000 deg,	P =   0.000 deg,	R =   90.000 deg
};
P[761]{
   GP1:
	UF : 0, UT : 6,		CONFIG : 'N U T, 0, 0, 0',
	X =  321.807  mm,	Y =   -128.838  mm,	Z =   -253.942  mm,
	W =  90.000 deg,	P =   0.000 deg,	R =   90.000 deg
};
P[762]{
   GP1:
	UF : 0, UT : 6,		CONFIG : 'N U T, 0, 0, 0',
	X =  319.900  mm,	Y =   -129.944  mm,	Z =   -253.951  mm,
	W =  90.000 deg,	P =   0.000 deg,	R =   90.000 deg
};
P[763]{
   GP1:
	UF : 0, UT : 6,		CONFIG : 'N U T, 0, 0, 0',
	X =  319.024  mm,	Y =   -130.324  mm,	Z =   -253.649  mm,
	W =  90.000 deg,	P =   0.000 deg,	R =   90.000 deg
};
P[764]{
   GP1:
	UF : 0, UT : 6,		CONFIG : 'N U T, 0, 0, 0',
	X =  316.387  mm,	Y =   -132.006  mm,	Z =   -254.033  mm,
	W =  90.000 deg,	P =   0.000 deg,	R =   90.000 deg
};
P[765]{
   GP1:
	UF : 0, UT : 6,		CONFIG : 'N U T, 0, 0, 0',
	X =  315.610  mm,	Y =   -132.481  mm,	Z =   -254.097  mm,
	W =  90.000 deg,	P =   0.000 deg,	R =   90.000 deg
};
P[766]{
   GP1:
	UF : 0, UT : 6,		CONFIG : 'N U T, 0, 0, 0',
	X =  311.873  mm,	Y =   -134.592  mm,	Z =   -253.985  mm,
	W =  90.000 deg,	P =   0.000 deg,	R =   90.000 deg
};
P[767]{
   GP1:
	UF : 0, UT : 6,		CONFIG : 'N U T, 0, 0, 0',
	X =  309.673  mm,	Y =   -135.866  mm,	Z =   -253.993  mm,
	W =  90.000 deg,	P =   0.000 deg,	R =   90.000 deg
};
P[768]{
   GP1:
	UF : 0, UT : 6,		CONFIG : 'N U T, 0, 0, 0',
	X =  308.744  mm,	Y =   -136.339  mm,	Z =   -253.841  mm,
	W =  90.000 deg,	P =   0.000 deg,	R =   90.000 deg
};
P[769]{
   GP1:
	UF : 0, UT : 6,		CONFIG : 'N U T, 0, 0, 0',
	X =  308.118  mm,	Y =   -136.658  mm,	Z =   -253.734  mm,
	W =  90.000 deg,	P =   0.000 deg,	R =   90.000 deg
};
P[770]{
   GP1:
	UF : 0, UT : 6,		CONFIG : 'N U T, 0, 0, 0',
	X =  307.321  mm,	Y =   -137.147  mm,	Z =   -253.808  mm,
	W =  90.000 deg,	P =   0.000 deg,	R =   90.000 deg
};
P[771]{
   GP1:
	UF : 0, UT : 6,		CONFIG : 'N U T, 0, 0, 0',
	X =  306.577  mm,	Y =   -137.581  mm,	Z =   -253.818  mm,
	W =  90.000 deg,	P =   0.000 deg,	R =   90.000 deg
};
P[772]{
   GP1:
	UF : 0, UT : 6,		CONFIG : 'N U T, 0, 0, 0',
	X =  305.696  mm,	Y =   -138.131  mm,	Z =   -253.920  mm,
	W =  90.000 deg,	P =   0.000 deg,	R =   90.000 deg
};
P[773]{
   GP1:
	UF : 0, UT : 6,		CONFIG : 'N U T, 0, 0, 0',
	X =  301.567  mm,	Y =   -140.409  mm,	Z =   -253.663  mm,
	W =  90.000 deg,	P =   0.000 deg,	R =   90.000 deg
};
P[774]{
   GP1:
	UF : 0, UT : 6,		CONFIG : 'N U T, 0, 0, 0',
	X =  299.698  mm,	Y =   -141.622  mm,	Z =   -253.984  mm,
	W =  90.000 deg,	P =   0.000 deg,	R =   90.000 deg
};
P[775]{
   GP1:
	UF : 0, UT : 6,		CONFIG : 'N U T, 0, 0, 0',
	X =  297.991  mm,	Y =   -142.593  mm,	Z =   -253.950  mm,
	W =  90.000 deg,	P =   0.000 deg,	R =   90.000 deg
};
P[776]{
   GP1:
	UF : 0, UT : 6,		CONFIG : 'N U T, 0, 0, 0',
	X =  296.523  mm,	Y =   -143.420  mm,	Z =   -253.901  mm,
	W =  90.000 deg,	P =   0.000 deg,	R =   90.000 deg
};
P[777]{
   GP1:
	UF : 0, UT : 6,		CONFIG : 'N U T, 0, 0, 0',
	X =  295.559  mm,	Y =   -144.058  mm,	Z =   -254.098  mm,
	W =  90.000 deg,	P =   0.000 deg,	R =   90.000 deg
};
P[778]{
   GP1:
	UF : 0, UT : 6,		CONFIG : 'N U T, 0, 0, 0',
	X =  294.961  mm,	Y =   -144.258  mm,	Z =   -253.743  mm,
	W =  90.000 deg,	P =   0.000 deg,	R =   90.000 deg
};
P[779]{
   GP1:
	UF : 0, UT : 6,		CONFIG : 'N U T, 0, 0, 0',
	X =  293.976  mm,	Y =   -144.930  mm,	Z =   -253.995  mm,
	W =  90.000 deg,	P =   0.000 deg,	R =   90.000 deg
};
P[780]{
   GP1:
	UF : 0, UT : 6,		CONFIG : 'N U T, 0, 0, 0',
	X =  291.089  mm,	Y =   -146.509  mm,	Z =   -253.782  mm,
	W =  90.000 deg,	P =   0.000 deg,	R =   90.000 deg
};
P[781]{
   GP1:
	UF : 0, UT : 6,		CONFIG : 'N U T, 0, 0, 0',
	X =  290.363  mm,	Y =   -146.952  mm,	Z =   -253.840  mm,
	W =  90.000 deg,	P =   0.000 deg,	R =   90.000 deg
};
P[782]{
   GP1:
	UF : 0, UT : 6,		CONFIG : 'N U T, 0, 0, 0',
	X =  288.474  mm,	Y =   -148.059  mm,	Z =   -253.877  mm,
	W =  90.000 deg,	P =   0.000 deg,	R =   90.000 deg
};
P[783]{
   GP1:
	UF : 0, UT : 6,		CONFIG : 'N U T, 0, 0, 0',
	X =  287.255  mm,	Y =   -148.665  mm,	Z =   -253.642  mm,
	W =  90.000 deg,	P =   0.000 deg,	R =   90.000 deg
};
P[784]{
   GP1:
	UF : 0, UT : 6,		CONFIG : 'N U T, 0, 0, 0',
	X =  285.502  mm,	Y =   -149.818  mm,	Z =   -253.985  mm,
	W =  90.000 deg,	P =   0.000 deg,	R =   90.000 deg
};
P[785]{
   GP1:
	UF : 0, UT : 6,		CONFIG : 'N U T, 0, 0, 0',
	X =  284.408  mm,	Y =   -150.373  mm,	Z =   -253.799  mm,
	W =  90.000 deg,	P =   0.000 deg,	R =   90.000 deg
};
P[786]{
   GP1:
	UF : 0, UT : 6,		CONFIG : 'N U T, 0, 0, 0',
	X =  283.563  mm,	Y =   -150.937  mm,	Z =   -253.982  mm,
	W =  90.000 deg,	P =   0.000 deg,	R =   90.000 deg
};
P[787]{
   GP1:
	UF : 0, UT : 6,		CONFIG : 'N U T, 0, 0, 0',
	X =  282.271  mm,	Y =   -151.728  mm,	Z =   -254.093  mm,
	W =  90.000 deg,	P =   0.000 deg,	R =   90.000 deg
};
P[788]{
   GP1:
	UF : 0, UT : 6,		CONFIG : 'N U T, 0, 0, 0',
	X =  281.313  mm,	Y =   -152.169  mm,	Z =   -253.819  mm,
	W =  90.000 deg,	P =   0.000 deg,	R =   90.000 deg
};
P[789]{
   GP1:
	UF : 0, UT : 6,		CONFIG : 'N U T, 0, 0, 0',
	X =  278.292  mm,	Y =   -153.964  mm,	Z =   -253.942  mm,
	W =  90.000 deg,	P =   0.000 deg,	R =   90.000 deg
};
P[790]{
   GP1:
	UF : 0, UT : 6,		CONFIG : 'N U T, 0, 0, 0',
	X =  277.478  mm,	Y =   -154.329  mm,	Z =   -253.689  mm,
	W =  90.000 deg,	P =   0.000 deg,	R =   90.000 deg
};
P[791]{
   GP1:
	UF : 0, UT : 6,		CONFIG : 'N U T, 0, 0, 0',
	X =  274.633  mm,	Y =   -156.044  mm,	Z =   -253.865  mm,
	W =  90.000 deg,	P =   0.000 deg,	R =   90.000 deg
};
P[792]{
   GP1:
	UF : 0, UT : 6,		CONFIG : 'N U T, 0, 0, 0',
	X =  269.148  mm,	Y =   -159.205  mm,	Z =   -253.847  mm,
	W =  90.000 deg,	P =   0.000 deg,	R =   90.000 deg
};
P[793]{
   GP1:
	UF : 0, UT : 6,		CONFIG : 'N U T, 0, 0, 0',
	X =  268.156  mm,	Y =   -159.870  mm,	Z =   -254.073  mm,
	W =  90.000 deg,	P =   0.000 deg,	R =   90.000 deg
};
P[794]{
   GP1:
	UF : 0, UT : 6,		CONFIG : 'N U T, 0, 0, 0',
	X =  267.180  mm,	Y =   -160.439  mm,	Z =   -254.086  mm,
	W =  90.000 deg,	P =   0.000 deg,	R =   90.000 deg
};
P[795]{
   GP1:
	UF : 0, UT : 6,		CONFIG : 'N U T, 0, 0, 0',
	X =  264.825  mm,	Y =   -161.805  mm,	Z =   -254.100  mm,
	W =  90.000 deg,	P =   0.000 deg,	R =   90.000 deg
};
P[796]{
   GP1:
	UF : 0, UT : 6,		CONFIG : 'N U T, 0, 0, 0',
	X =  261.286  mm,	Y =   -163.727  mm,	Z =   -253.806  mm,
	W =  90.000 deg,	P =   0.000 deg,	R =   90.000 deg
};
P[797]{
   GP1:
	UF : 0, UT : 6,		CONFIG : 'N U T, 0, 0, 0',
	X =  260.130  mm,	Y =   -164.411  mm,	Z =   -253.845  mm,
	W =  90.000 deg,	P =   0.000 deg,	R =   90.000 deg
};
P[798]{
   GP1:
	UF : 0, UT : 6,		CONFIG : 'N U T, 0, 0, 0',
	X =  258.513  mm,	Y =   -165.388  mm,	Z =   -253.951  mm,
	W =  90.000 deg,	P =   0.000 deg,	R =   90.000 deg
};
P[799]{
   GP1:
	UF : 0, UT : 6,		CONFIG : 'N U T, 0, 0, 0',
	X =  257.805  mm,	Y =   -165.711  mm,	Z =   -253.744  mm,
	W =  90.000 deg,	P =   0.000 deg,	R =   90.000 deg
};
P[800]{
   GP1:
	UF : 0, UT : 6,		CONFIG : 'N U T, 0, 0, 0',
	X =  255.152  mm,	Y =   -167.362  mm,	Z =   -254.034  mm,
	W =  90.000 deg,	P =   0.000 deg,	R =   90.000 deg
};
P[801]{
   GP1:
	UF : 0, UT : 6,		CONFIG : 'N U T, 0, 0, 0',
	X =  251.444  mm,	Y =   -169.541  mm,	Z =   -254.124  mm,
	W =  90.000 deg,	P =   0.000 deg,	R =   90.000 deg
};
P[802]{
   GP1:
	UF : 0, UT : 6,		CONFIG : 'N U T, 0, 0, 0',
	X =  249.911  mm,	Y =   -170.307  mm,	Z =   -253.837  mm,
	W =  90.000 deg,	P =   0.000 deg,	R =   90.000 deg
};
P[803]{
   GP1:
	UF : 0, UT : 6,		CONFIG : 'N U T, 0, 0, 0',
	X =  249.132  mm,	Y =   -170.706  mm,	Z =   -253.714  mm,
	W =  90.000 deg,	P =   0.000 deg,	R =   90.000 deg
};
P[804]{
   GP1:
	UF : 0, UT : 6,		CONFIG : 'N U T, 0, 0, 0',
	X =  248.500  mm,	Y =   -171.043  mm,	Z =   -253.644  mm,
	W =  90.000 deg,	P =   0.000 deg,	R =   90.000 deg
};
P[805]{
   GP1:
	UF : 0, UT : 6,		CONFIG : 'N U T, 0, 0, 0',
	X =  247.897  mm,	Y =   -171.500  mm,	Z =   -253.906  mm,
	W =  90.000 deg,	P =   0.000 deg,	R =   90.000 deg
};
P[806]{
   GP1:
	UF : 0, UT : 6,		CONFIG : 'N U T, 0, 0, 0',
	X =  245.882  mm,	Y =   -172.747  mm,	Z =   -254.112  mm,
	W =  90.000 deg,	P =   0.000 deg,	R =   90.000 deg
};
P[807]{
   GP1:
	UF : 0, UT : 6,		CONFIG : 'N U T, 0, 0, 0',
	X =  244.972  mm,	Y =   -173.274  mm,	Z =   -254.116  mm,
	W =  90.000 deg,	P =   0.000 deg,	R =   90.000 deg
};
P[808]{
   GP1:
	UF : 0, UT : 6,		CONFIG : 'N U T, 0, 0, 0',
	X =  243.429  mm,	Y =   -174.097  mm,	Z =   -253.949  mm,
	W =  90.000 deg,	P =   0.000 deg,	R =   90.000 deg
};
P[809]{
   GP1:
	UF : 0, UT : 6,		CONFIG : 'N U T, 0, 0, 0',
	X =  241.658  mm,	Y =   -175.002  mm,	Z =   -253.665  mm,
	W =  90.000 deg,	P =   0.000 deg,	R =   90.000 deg
};
P[810]{
   GP1:
	UF : 0, UT : 6,		CONFIG : 'N U T, 0, 0, 0',
	X =  238.813  mm,	Y =   -176.761  mm,	Z =   -253.948  mm,
	W =  90.000 deg,	P =   0.000 deg,	R =   90.000 deg
};
P[811]{
   GP1:
	UF : 0, UT : 6,		CONFIG : 'N U T, 0, 0, 0',
	X =  235.699  mm,	Y =   -178.484  mm,	Z =   -253.764  mm,
	W =  90.000 deg,	P =   0.000 deg,	R =   90.000 deg
};
P[812]{
   GP1:
	UF : 0, UT : 6,		CONFIG : 'N U T, 0, 0, 0',
	X =  233.292  mm,	Y =   -179.923  mm,	Z =   -253.886  mm,
	W =  90.000 deg,	P =   0.000 deg,	R =   90.000 deg
};
P[813]{
   GP1:
	UF : 0, UT : 6,		CONFIG : 'N U T, 0, 0, 0',
	X =  231.929  mm,	Y =   -180.702  mm,	Z =   -253.867  mm,
	W =  90.000 deg,	P =   0.000 deg,	R =   90.000 deg
};
P[814]{
   GP1:
	UF : 0, UT : 6,		CONFIG : 'N U T, 0, 0, 0',
	X =  230.471  mm,	Y =   -181.552  mm,	Z =   -253.887  mm,
	W =  90.000 deg,	P =   0.000 deg,	R =   90.000 deg
};
P[815]{
   GP1:
	UF : 0, UT : 6,		CONFIG : 'N U T, 0, 0, 0',
	X =  229.536  mm,	Y =   -182.143  mm,	Z =   -254.011  mm,
	W =  90.000 deg,	P =   0.000 deg,	R =   90.000 deg
};
P[816]{
   GP1:
	UF : 0, UT : 6,		CONFIG : 'N U T, 0, 0, 0',
	X =  226.591  mm,	Y =   -183.728  mm,	Z =   -253.730  mm,
	W =  90.000 deg,	P =   0.000 deg,	R =   90.000 deg
};
P[817]{
   GP1:
	UF : 0, UT : 6,		CONFIG : 'N U T, 0, 0, 0',
	X =  225.117  mm,	Y =   -184.627  mm,	Z =   -253.845  mm,
	W =  90.000 deg,	P =   0.000 deg,	R =   90.000 deg
};
P[818]{
   GP1:
	UF : 0, UT : 6,		CONFIG : 'N U T, 0, 0, 0',
	X =  223.881  mm,	Y =   -185.356  mm,	Z =   -253.884  mm,
	W =  90.000 deg,	P =   0.000 deg,	R =   90.000 deg
};
P[819]{
   GP1:
	UF : 0, UT : 6,		CONFIG : 'N U T, 0, 0, 0',
	X =  221.079  mm,	Y =   -186.929  mm,	Z =   -253.774  mm,
	W =  90.000 deg,	P =   0.000 deg,	R =   90.000 deg
};
P[820]{
   GP1:
	UF : 0, UT : 6,		CONFIG : 'N U T, 0, 0, 0',
	X =  218.861  mm,	Y =   -188.297  mm,	Z =   -253.984  mm,
	W =  90.000 deg,	P =   0.000 deg,	R =   90.000 deg
};
P[821]{
   GP1:
	UF : 0, UT : 6,		CONFIG : 'N U T, 0, 0, 0',
	X =  218.137  mm,	Y =   -188.653  mm,	Z =   -253.837  mm,
	W =  90.000 deg,	P =   0.000 deg,	R =   90.000 deg
};
P[822]{
   GP1:
	UF : 0, UT : 6,		CONFIG : 'N U T, 0, 0, 0',
	X =  214.673  mm,	Y =   -190.740  mm,	Z =   -254.047  mm,
	W =  90.000 deg,	P =   0.000 deg,	R =   90.000 deg
};
P[823]{
   GP1:
	UF : 0, UT : 6,		CONFIG : 'N U T, 0, 0, 0',
	X =  212.315  mm,	Y =   -191.943  mm,	Z =   -253.662  mm,
	W =  90.000 deg,	P =   0.000 deg,	R =   90.000 deg
};
P[824]{
   GP1:
	UF : 0, UT : 6,		CONFIG : 'N U T, 0, 0, 0',
	X =  207.810  mm,	Y =   -194.640  mm,	Z =   -253.896  mm,
	W =  90.000 deg,	P =   0.000 deg,	R =   90.000 deg
};
P[825]{
   GP1:
	UF : 0, UT : 6,		CONFIG : 'N U T, 0, 0, 0',
	X =  206.764  mm,	Y =   -195.313  mm,	Z =   -254.063  mm,
	W =  90.000 deg,	P =   0.000 deg,	R =   90.000 deg
};
P[826]{
   GP1:
	UF : 0, UT : 6,		CONFIG : 'N U T, 0, 0, 0',
	X =  204.894  mm,	Y =   -196.234  mm,	Z =   -253.676  mm,
	W =  90.000 deg,	P =   0.000 deg,	R =   90.000 deg
};
P[827]{
   GP1:
	UF : 0, UT : 6,		CONFIG : 'N U T, 0, 0, 0',
	X =  203.897  mm,	Y =   -196.932  mm,	Z =   -253.975  mm,
	W =  90.000 deg,	P =   0.000 deg,	R =   90.000 deg
};
P[828]{
   GP1:
	UF : 0, UT : 6,		CONFIG : 'N U T, 0, 0, 0',
	X =  202.830  mm,	Y =   -197.513  mm,	Z =   -253.890  mm,
	W =  90.000 deg,	P =   0.000 deg,	R =   90.000 deg
};
P[829]{
   GP1:
	UF : 0, UT : 6,		CONFIG : 'N U T, 0, 0, 0',
	X =  201.232  mm,	Y =   -198.443  mm,	Z =   -253.909  mm,
	W =  90.000 deg,	P =   0.000 deg,	R =   90.000 deg
};
P[830]{
   GP1:
	UF : 0, UT : 6,		CONFIG : 'N U T, 0, 0, 0',
	X =  198.409  mm,	Y =   -200.090  mm,	Z =   -253.947  mm,
	W =  90.000 deg,	P =   0.000 deg,	R =   90.000 deg
};
P[831]{
   GP1:
	UF : 0, UT : 6,		CONFIG : 'N U T, 0, 0, 0',
	X =  196.428  mm,	Y =   -201.215  mm,	Z =   -253.903  mm,
	W =  90.000 deg,	P =   0.000 deg,	R =   90.000 deg
};
P[832]{
   GP1:
	UF : 0, UT : 6,		CONFIG : 'N U T, 0, 0, 0',
	X =  192.774  mm,	Y =   -203.290  mm,	Z =   -253.818  mm,
	W =  90.000 deg,	P =   0.000 deg,	R =   90.000 deg
};
P[833]{
   GP1:
	UF : 0, UT : 6,		CONFIG : 'N U T, 0, 0, 0',
	X =  190.073  mm,	Y =   -204.821  mm,	Z =   -253.749  mm,
	W =  90.000 deg,	P =   0.000 deg,	R =   90.000 deg
};
P[834]{
   GP1:
	UF : 0, UT : 6,		CONFIG : 'N U T, 0, 0, 0',
	X =  189.259  mm,	Y =   -205.314  mm,	Z =   -253.804  mm,
	W =  90.000 deg,	P =   0.000 deg,	R =   90.000 deg
};
P[835]{
   GP1:
	UF : 0, UT : 6,		CONFIG : 'N U T, 0, 0, 0',
	X =  188.481  mm,	Y =   -205.790  mm,	Z =   -253.868  mm,
	W =  90.000 deg,	P =   0.000 deg,	R =   90.000 deg
};
P[836]{
   GP1:
	UF : 0, UT : 6,		CONFIG : 'N U T, 0, 0, 0',
	X =  187.376  mm,	Y =   -206.355  mm,	Z =   -253.692  mm,
	W =  90.000 deg,	P =   0.000 deg,	R =   90.000 deg
};
P[837]{
   GP1:
	UF : 0, UT : 6,		CONFIG : 'N U T, 0, 0, 0',
	X =  184.558  mm,	Y =   -208.154  mm,	Z =   -254.110  mm,
	W =  90.000 deg,	P =   0.000 deg,	R =   90.000 deg
};
P[838]{
   GP1:
	UF : 0, UT : 6,		CONFIG : 'N U T, 0, 0, 0',
	X =  183.569  mm,	Y =   -208.541  mm,	Z =   -253.664  mm,
	W =  90.000 deg,	P =   0.000 deg,	R =   90.000 deg
};
P[839]{
   GP1:
	UF : 0, UT : 6,		CONFIG : 'N U T, 0, 0, 0',
	X =  182.338  mm,	Y =   -209.334  mm,	Z =   -253.861  mm,
	W =  90.000 deg,	P =   0.000 deg,	R =   90.000 deg
};
P[840]{
   GP1:
	UF : 0, UT : 6,		CONFIG : 'N U T, 0, 0, 0',
	X =  180.736  mm,	Y =   -210.340  mm,	Z =   -254.060  mm,
	W =  90.000 deg,	P =   0.000 deg,	R =   90.000 deg
};
P[841]{
   GP1:
	UF : 0, UT : 6,		CONFIG : 'N U T, 0, 0, 0',
	X =  179.732  mm,	Y =   -210.849  mm,	Z =   -253.885  mm,
	W =  90.000 deg,	P =   0.000 deg,	R =   90.000 deg
};
P[842]{
   GP1:
	UF : 0, UT : 6,		CONFIG : 'N U T, 0, 0, 0',
	X =  177.168  mm,	Y =   -212.411  mm,	Z =   -254.087  mm,
	W =  90.000 deg,	P =   0.000 deg,	R =   90.000 deg
};
P[843]{
   GP1:
	UF : 0, UT : 6,		CONFIG : 'N U T, 0, 0, 0',
	X =  176.287  mm,	Y =   -212.921  mm,	Z =   -254.089  mm,
	W =  90.000 deg,	P =   0.000 deg,	R =   90.000 deg
};
P[844]{
   GP1:
	UF : 0, UT : 6,		CONFIG : 'N U T, 0, 0, 0',
	X =  172.206  mm,	Y =   -215.212  mm,	Z =   -253.929  mm,
	W =  90.000 deg,	P =   0.000 deg,	R =   90.000 deg
};
P[845]{
   GP1:
	UF : 0, UT : 6,		CONFIG : 'N U T, 0, 0, 0',
	X =  168.566  mm,	Y =   -217.314  mm,	Z =   -253.931  mm,
	W =  90.000 deg,	P =   0.000 deg,	R =   90.000 deg
};
P[846]{
   GP1:
	UF : 0, UT : 6,		CONFIG : 'N U T, 0, 0, 0',
	X =  167.110  mm,	Y =   -218.075  mm,	Z =   -253.737  mm,
	W =  90.000 deg,	P =   0.000 deg,	R =   90.000 deg
};
P[847]{
   GP1:
	UF : 0, UT : 6,		CONFIG : 'N U T, 0, 0, 0',
	X =  164.088  mm,	Y =   -219.949  mm,	Z =   -254.051  mm,
	W =  90.000 deg,	P =   0.000 deg,	R =   90.000 deg
};
P[848]{
   GP1:
	UF : 0, UT : 6,		CONFIG : 'N U T, 0, 0, 0',
	X =  163.241  mm,	Y =   -220.329  mm,	Z =   -253.787  mm,
	W =  90.000 deg,	P =   0.000 deg,	R =   90.000 deg
};
P[849]{
   GP1:
	UF : 0, UT : 6,		CONFIG : 'N U T, 0, 0, 0',
	X =  161.377  mm,	Y =   -221.407  mm,	Z =   -253.790  mm,
	W =  90.000 deg,	P =   0.000 deg,	R =   90.000 deg
};
P[850]{
   GP1:
	UF : 0, UT : 6,		CONFIG : 'N U T, 0, 0, 0',
	X =  157.951  mm,	Y =   -223.395  mm,	Z =   -253.813  mm,
	W =  90.000 deg,	P =   0.000 deg,	R =   90.000 deg
};
P[851]{
   GP1:
	UF : 0, UT : 6,		CONFIG : 'N U T, 0, 0, 0',
	X =  157.320  mm,	Y =   -223.740  mm,	Z =   -253.767  mm,
	W =  90.000 deg,	P =   0.000 deg,	R =   90.000 deg
};
P[852]{
   GP1:
	UF : 0, UT : 6,		CONFIG : 'N U T, 0, 0, 0',
	X =  154.731  mm,	Y =   -225.257  mm,	Z =   -253.821  mm,
	W =  90.000 deg,	P =   0.000 deg,	R =   90.000 deg
};
P[853]{
   GP1:
	UF : 0, UT : 6,		CONFIG : 'N U T, 0, 0, 0',
	X =  154.070  mm,	Y =   -225.724  mm,	Z =   -254.028  mm,
	W =  90.000 deg,	P =   0.000 deg,	R =   90.000 deg
};
P[854]{
   GP1:
	UF : 0, UT : 6,		CONFIG : 'N U T, 0, 0, 0',
	X =  151.415  mm,	Y =   -227.245  mm,	Z =   -253.999  mm,
	W =  90.000 deg,	P =   0.000 deg,	R =   90.000 deg
};
P[855]{
   GP1:
	UF : 0, UT : 6,		CONFIG : 'N U T, 0, 0, 0',
	X =  148.299  mm,	Y =   -228.971  mm,	Z =   -253.819  mm,
	W =  90.000 deg,	P =   0.000 deg,	R =   90.000 deg
};
P[856]{
   GP1:
	UF : 0, UT : 6,		CONFIG : 'N U T, 0, 0, 0',
	X =  147.650  mm,	Y =   -229.469  mm,	Z =   -254.119  mm,
	W =  90.000 deg,	P =   0.000 deg,	R =   90.000 deg
};
P[857]{
   GP1:
	UF : 0, UT : 6,		CONFIG : 'N U T, 0, 0, 0',
	X =  145.597  mm,	Y =   -230.542  mm,	Z =   -253.848  mm,
	W =  90.000 deg,	P =   0.000 deg,	R =   90.000 deg
};
P[858]{
   GP1:
	UF : 0, UT : 6,		CONFIG : 'N U T, 0, 0, 0',
	X =  144.044  mm,	Y =   -231.506  mm,	Z =   -254.012  mm,
	W =  90.000 deg,	P =   0.000 deg,	R =   90.000 deg
};
P[859]{
   GP1:
	UF : 0, UT : 6,		CONFIG : 'N U T, 0, 0, 0',
	X =  141.837  mm,	Y =   -232.783  mm,	Z =   -254.018  mm,
	W =  90.000 deg,	P =   0.000 deg,	R =   90.000 deg
};
P[860]{
   GP1:
	UF : 0, UT : 6,		CONFIG : 'N U T, 0, 0, 0',
	X =  141.133  mm,	Y =   -233.229  mm,	Z =   -254.115  mm,
	W =  90.000 deg,	P =   0.000 deg,	R =   90.000 deg
};
P[861]{
   GP1:
	UF : 0, UT : 6,		CONFIG : 'N U T, 0, 0, 0',
	X =  138.869  mm,	Y =   -234.366  mm,	Z =   -253.700  mm,
	W =  90.000 deg,	P =   0.000 deg,	R =   90.000 deg
};
P[862]{
   GP1:
	UF : 0, UT : 6,		CONFIG : 'N U T, 0, 0, 0',
	X =  137.735  mm,	Y =   -235.031  mm,	Z =   -253.724  mm,
	W =  90.000 deg,	P =   0.000 deg,	R =   90.000 deg
};
P[863]{
   GP1:
	UF : 0, UT : 6,		CONFIG : 'N U T, 0, 0, 0',
	X =  136.027  mm,	Y =   -236.182  mm,	Z =   -254.126  mm,
	W =  90.000 deg,	P =   0.000 deg,	R =   90.000 deg
};
P[864]{
   GP1:
	UF : 0, UT : 6,		CONFIG : 'N U T, 0, 0, 0',
	X =  134.627  mm,	Y =   -236.859  mm,	Z =   -253.807  mm,
	W =  90.000 deg,	P =   0.000 deg,	R =   90.000 deg
};
P[865]{
   GP1:
	UF : 0, UT : 6,		CONFIG : 'N U T, 0, 0, 0',
	X =  133.920  mm,	Y =   -237.347  mm,	Z =   -254.000  mm,
	W =  90.000 deg,	P =   0.000 deg,	R =   90.000 deg
};
P[866]{
   GP1:
	UF : 0, UT : 6,		CONFIG : 'N U T, 0, 0, 0',
	X =  131.505  mm,	Y =   -238.791  mm,	Z =   -254.122  mm,
	W =  90.000 deg,	P =   0.000 deg,	R =   90.000 deg
};
P[867]{
   GP1:
	UF : 0, UT : 6,		CONFIG : 'N U T, 0, 0, 0',
	X =  130.307  mm,	Y =   -239.460  mm,	Z =   -254.064  mm,
	W =  90.000 deg,	P =   0.000 deg,	R =   90.000 deg
};
P[868]{
   GP1:
	UF : 0, UT : 6,		CONFIG : 'N U T, 0, 0, 0',
	X =  129.409  mm,	Y =   -239.837  mm,	Z =   -253.723  mm,
	W =  90.000 deg,	P =   0.000 deg,	R =   90.000 deg
};
P[869]{
   GP1:
	UF : 0, UT : 6,		CONFIG : 'N U T, 0, 0, 0',
	X =  128.464  mm,	Y =   -240.351  mm,	Z =   -253.644  mm,
	W =  90.000 deg,	P =   0.000 deg,	R =   90.000 deg
};
P[870]{
   GP1:
	UF : 0, UT : 6,		CONFIG : 'N U T, 0, 0, 0',
	X =  127.453  mm,	Y =   -241.056  mm,	Z =   -253.939  mm,
	W =  90.000 deg,	P =   0.000 deg,	R =   90.000 deg
};
P[871]{
   GP1:
	UF : 0, UT : 6,		CONFIG : 'N U T, 0, 0, 0',
	X =  124.164  mm,	Y =   -243.017  mm,	Z =   -254.088  mm,
	W =  90.000 deg,	P =   0.000 deg,	R =   90.000 deg
};
P[872]{
   GP1:
	UF : 0, UT : 6,		CONFIG : 'N U T, 0, 0, 0',
	X =  123.509  mm,	Y =   -243.264  mm,	Z =   -253.770  mm,
	W =  90.000 deg,	P =   0.000 deg,	R =   90.000 deg
};
P[873]{
   GP1:
	UF : 0, UT : 6,		CONFIG : 'N U T, 0, 0, 0',
	X =  121.257  mm,	Y =   -244.707  mm,	Z =   -254.117  mm,
	W =  90.000 deg,	P =   0.000 deg,	R =   90.000 deg
};
P[874]{
   GP1:
	UF : 0, UT : 6,		CONFIG : 'N U T, 0, 0, 0',
	X =  117.331  mm,	Y =   -246.778  mm,	Z =   -253.641  mm,
	W =  90.000 deg,	P =   0.000 deg,	R =   90.000 deg
};
P[875]{
   GP1:
	UF : 0, UT : 6,		CONFIG : 'N U T, 0, 0, 0',
	X =  116.333  mm,	Y =   -247.396  mm,	Z =   -253.745  mm,
	W =  90.000 deg,	P =   0.000 deg,	R =   90.000 deg
};
P[876]{
   GP1:
	UF : 0, UT : 6,		CONFIG : 'N U T, 0, 0, 0',
	X =  115.503  mm,	Y =   -247.928  mm,	Z =   -253.873  mm,
	W =  90.000 deg,	P =   0.000 deg,	R =   90.000 deg
};
P[877]{
   GP1:
	UF : 0, UT : 6,		CONFIG : 'N U T, 0, 0, 0',
	X =  114.923  mm,	Y =   -248.304  mm,	Z =   -253.971  mm,
	W =  90.000 deg,	P =   0.000 deg,	R =   90.000 deg
};
P[878]{
   GP1:
	UF : 0, UT : 6,		CONFIG : 'N U T, 0, 0, 0',
	X =  114.292  mm,	Y =   -248.660  mm,	Z =   -253.953  mm,
	W =  90.000 deg,	P =   0.000 deg,	R =   90.000 deg
};
P[879]{
   GP1:
	UF : 0, UT : 6,		CONFIG : 'N U T, 0, 0, 0',
	X =  113.519  mm,	Y =   -249.081  mm,	Z =   -253.889  mm,
	W =  90.000 deg,	P =   0.000 deg,	R =   90.000 deg
};
P[880]{
   GP1:
	UF : 0, UT : 6,		CONFIG : 'N U T, 0, 0, 0',
	X =  112.836  mm,	Y =   -249.508  mm,	Z =   -253.969  mm,
	W =  90.000 deg,	P =   0.000 deg,	R =   90.000 deg
};
P[881]{
   GP1:
	UF : 0, UT : 6,		CONFIG : 'N U T, 0, 0, 0',
	X =  112.040  mm,	Y =   -249.896  mm,	Z =   -253.796  mm,
	W =  90.000 deg,	P =   0.000 deg,	R =   90.000 deg
};
P[882]{
   GP1:
	UF : 0, UT : 6,		CONFIG : 'N U T, 0, 0, 0',
	X =  111.234  mm,	Y =   -250.453  mm,	Z =   -254.017  mm,
	W =  90.000 deg,	P =   0.000 deg,	R =   90.000 deg
};
P[883]{
   GP1:
	UF : 0, UT : 6,		CONFIG : 'N U T, 0, 0, 0',
	X =  110.587  mm,	Y =   -250.813  mm,	Z =   -253.986  mm,
	W =  90.000 deg,	P =   0.000 deg,	R =   90.000 deg
};
P[884]{
   GP1:
	UF : 0, UT : 6,		CONFIG : 'N U T, 0, 0, 0',
	X =  108.548  mm,	Y =   -251.967  mm,	Z =   -253.927  mm,
	W =  90.000 deg,	P =   0.000 deg,	R =   90.000 deg
};
P[885]{
   GP1:
	UF : 0, UT : 6,		CONFIG : 'N U T, 0, 0, 0',
	X =  106.804  mm,	Y =   -252.909  mm,	Z =   -253.770  mm,
	W =  90.000 deg,	P =   0.000 deg,	R =   90.000 deg
};
P[886]{
   GP1:
	UF : 0, UT : 6,		CONFIG : 'N U T, 0, 0, 0',
	X =  103.477  mm,	Y =   -252.496  mm,	Z =   -248.105  mm,
	W =  90.000 deg,	P =   0.000 deg,	R =   90.000 deg
};
P[887]{
   GP1:
	UF : 0, UT : 6,		CONFIG : 'N U T, 0, 0, 0',
	X =  102.427  mm,	Y =   -253.131  mm,	Z =   -248.175  mm,
	W =  90.000 deg,	P =   0.000 deg,	R =   90.000 deg
};
P[888]{
   GP1:
	UF : 0, UT : 6,		CONFIG : 'N U T, 0, 0, 0',
	X =  101.793  mm,	Y =   -253.342  mm,	Z =   -247.800  mm,
	W =  90.000 deg,	P =   0.000 deg,	R =   90.000 deg
};
P[889]{
   GP1:
	UF : 0, UT : 6,		CONFIG : 'N U T, 0, 0, 0',
	X =  99.755  mm,	Y =   -254.566  mm,	Z =   -247.914  mm,
	W =  90.000 deg,	P =   0.000 deg,	R =   90.000 deg
};
P[890]{
   GP1:
	UF : 0, UT : 6,		CONFIG : 'N U T, 0, 0, 0',
	X =  97.303  mm,	Y =   -256.053  mm,	Z =   -248.085  mm,
	W =  90.000 deg,	P =   0.000 deg,	R =   90.000 deg
};
P[891]{
   GP1:
	UF : 0, UT : 6,		CONFIG : 'N U T, 0, 0, 0',
	X =  96.088  mm,	Y =   -256.663  mm,	Z =   -247.865  mm,
	W =  90.000 deg,	P =   0.000 deg,	R =   90.000 deg
};
P[892]{
   GP1:
	UF : 0, UT : 6,		CONFIG : 'N U T, 0, 0, 0',
	X =  94.760  mm,	Y =   -257.401  mm,	Z =   -247.796  mm,
	W =  90.000 deg,	P =   0.000 deg,	R =   90.000 deg
};
P[893]{
   GP1:
	UF : 0, UT : 6,		CONFIG : 'N U T, 0, 0, 0',
	X =  91.348  mm,	Y =   -259.498  mm,	Z =   -248.103  mm,
	W =  90.000 deg,	P =   0.000 deg,	R =   90.000 deg
};
P[894]{
   GP1:
	UF : 0, UT : 6,		CONFIG : 'N U T, 0, 0, 0',
	X =  90.367  mm,	Y =   -259.960  mm,	Z =   -247.849  mm,
	W =  90.000 deg,	P =   0.000 deg,	R =   90.000 deg
};
P[895]{
   GP1:
	UF : 0, UT : 6,		CONFIG : 'N U T, 0, 0, 0',
	X =  89.072  mm,	Y =   -260.853  mm,	Z =   -248.201  mm,
	W =  90.000 deg,	P =   0.000 deg,	R =   90.000 deg
};
P[896]{
   GP1:
	UF : 0, UT : 6,		CONFIG : 'N U T, 0, 0, 0',
	X =  87.501  mm,	Y =   -261.651  mm,	Z =   -247.938  mm,
	W =  90.000 deg,	P =   0.000 deg,	R =   90.000 deg
};
P[897]{
   GP1:
	UF : 0, UT : 6,		CONFIG : 'N U T, 0, 0, 0',
	X =  86.385  mm,	Y =   -262.290  mm,	Z =   -247.923  mm,
	W =  90.000 deg,	P =   0.000 deg,	R =   90.000 deg
};
P[898]{
   GP1:
	UF : 0, UT : 6,		CONFIG : 'N U T, 0, 0, 0',
	X =  85.363  mm,	Y =   -262.914  mm,	Z =   -248.006  mm,
	W =  90.000 deg,	P =   0.000 deg,	R =   90.000 deg
};
P[899]{
   GP1:
	UF : 0, UT : 6,		CONFIG : 'N U T, 0, 0, 0',
	X =  84.586  mm,	Y =   -263.268  mm,	Z =   -247.776  mm,
	W =  90.000 deg,	P =   0.000 deg,	R =   90.000 deg
};
P[900]{
   GP1:
	UF : 0, UT : 6,		CONFIG : 'N U T, 0, 0, 0',
	X =  81.251  mm,	Y =   -265.207  mm,	Z =   -247.808  mm,
	W =  90.000 deg,	P =   0.000 deg,	R =   90.000 deg
};
P[901]{
   GP1:
	UF : 0, UT : 6,		CONFIG : 'N U T, 0, 0, 0',
	X =  80.556  mm,	Y =   -265.774  mm,	Z =   -248.211  mm,
	W =  90.000 deg,	P =   0.000 deg,	R =   90.000 deg
};
P[902]{
   GP1:
	UF : 0, UT : 6,		CONFIG : 'N U T, 0, 0, 0',
	X =  79.541  mm,	Y =   -266.195  mm,	Z =   -247.812  mm,
	W =  90.000 deg,	P =   0.000 deg,	R =   90.000 deg
};
P[903]{
   GP1:
	UF : 0, UT : 6,		CONFIG : 'N U T, 0, 0, 0',
	X =  78.115  mm,	Y =   -267.008  mm,	Z =   -247.788  mm,
	W =  90.000 deg,	P =   0.000 deg,	R =   90.000 deg
};
P[904]{
   GP1:
	UF : 0, UT : 6,		CONFIG : 'N U T, 0, 0, 0',
	X =  77.186  mm,	Y =   -267.696  mm,	Z =   -248.154  mm,
	W =  90.000 deg,	P =   0.000 deg,	R =   90.000 deg
};
P[905]{
   GP1:
	UF : 0, UT : 6,		CONFIG : 'N U T, 0, 0, 0',
	X =  73.898  mm,	Y =   -269.557  mm,	Z =   -248.065  mm,
	W =  90.000 deg,	P =   0.000 deg,	R =   90.000 deg
};
P[906]{
   GP1:
	UF : 0, UT : 6,		CONFIG : 'N U T, 0, 0, 0',
	X =  72.084  mm,	Y =   -270.539  mm,	Z =   -247.905  mm,
	W =  90.000 deg,	P =   0.000 deg,	R =   90.000 deg
};
P[907]{
   GP1:
	UF : 0, UT : 6,		CONFIG : 'N U T, 0, 0, 0',
	X =  70.657  mm,	Y =   -271.456  mm,	Z =   -248.129  mm,
	W =  90.000 deg,	P =   0.000 deg,	R =   90.000 deg
};
P[908]{
   GP1:
	UF : 0, UT : 6,		CONFIG : 'N U T, 0, 0, 0',
	X =  67.795  mm,	Y =   -273.149  mm,	Z =   -248.229  mm,
	W =  90.000 deg,	P =   0.000 deg,	R =   90.000 deg
};
P[909]{
   GP1:
	UF : 0, UT : 6,		CONFIG : 'N U T, 0, 0, 0',
	X =  67.043  mm,	Y =   -273.536  mm,	Z =   -248.112  mm,
	W =  90.000 deg,	P =   0.000 deg,	R =   90.000 deg
};
P[910]{
   GP1:
	UF : 0, UT : 6,		CONFIG : 'N U T, 0, 0, 0',
	X =  66.413  mm,	Y =   -273.811  mm,	Z =   -247.900  mm,
	W =  90.000 deg,	P =   0.000 deg,	R =   90.000 deg
};
P[911]{
   GP1:
	UF : 0, UT : 6,		CONFIG : 'N U T, 0, 0, 0',
	X =  64.975  mm,	Y =   -274.681  mm,	Z =   -247.996  mm,
	W =  90.000 deg,	P =   0.000 deg,	R =   90.000 deg
};
P[912]{
   GP1:
	UF : 0, UT : 6,		CONFIG : 'N U T, 0, 0, 0',
	X =  63.850  mm,	Y =   -275.257  mm,	Z =   -247.817  mm,
	W =  90.000 deg,	P =   0.000 deg,	R =   90.000 deg
};
P[913]{
   GP1:
	UF : 0, UT : 6,		CONFIG : 'N U T, 0, 0, 0',
	X =  61.562  mm,	Y =   -276.714  mm,	Z =   -248.145  mm,
	W =  90.000 deg,	P =   0.000 deg,	R =   90.000 deg
};
P[914]{
   GP1:
	UF : 0, UT : 6,		CONFIG : 'N U T, 0, 0, 0',
	X =  60.307  mm,	Y =   -277.318  mm,	Z =   -247.854  mm,
	W =  90.000 deg,	P =   0.000 deg,	R =   90.000 deg
};
P[915]{
   GP1:
	UF : 0, UT : 6,		CONFIG : 'N U T, 0, 0, 0',
	X =  58.562  mm,	Y =   -278.453  mm,	Z =   -248.164  mm,
	W =  90.000 deg,	P =   0.000 deg,	R =   90.000 deg
};
P[916]{
   GP1:
	UF : 0, UT : 6,		CONFIG : 'N U T, 0, 0, 0',
	X =  57.669  mm,	Y =   -278.933  mm,	Z =   -248.078  mm,
	W =  90.000 deg,	P =   0.000 deg,	R =   90.000 deg
};
P[917]{
   GP1:
	UF : 0, UT : 6,		CONFIG : 'N U T, 0, 0, 0',
	X =  56.915  mm,	Y =   -279.286  mm,	Z =   -247.877  mm,
	W =  90.000 deg,	P =   0.000 deg,	R =   90.000 deg
};
P[918]{
   GP1:
	UF : 0, UT : 6,		CONFIG : 'N U T, 0, 0, 0',
	X =  54.017  mm,	Y =   -280.941  mm,	Z =   -247.833  mm,
	W =  90.000 deg,	P =   0.000 deg,	R =   90.000 deg
};
P[919]{
   GP1:
	UF : 0, UT : 6,		CONFIG : 'N U T, 0, 0, 0',
	X =  50.052  mm,	Y =   -283.362  mm,	Z =   -248.152  mm,
	W =  90.000 deg,	P =   0.000 deg,	R =   90.000 deg
};
P[920]{
   GP1:
	UF : 0, UT : 6,		CONFIG : 'N U T, 0, 0, 0',
	X =  47.821  mm,	Y =   -284.622  mm,	Z =   -248.083  mm,
	W =  90.000 deg,	P =   0.000 deg,	R =   90.000 deg
};
P[921]{
   GP1:
	UF : 0, UT : 6,		CONFIG : 'N U T, 0, 0, 0',
	X =  46.365  mm,	Y =   -285.410  mm,	Z =   -247.956  mm,
	W =  90.000 deg,	P =   0.000 deg,	R =   90.000 deg
};
P[922]{
   GP1:
	UF : 0, UT : 6,		CONFIG : 'N U T, 0, 0, 0',
	X =  42.959  mm,	Y =   -287.385  mm,	Z =   -247.976  mm,
	W =  90.000 deg,	P =   0.000 deg,	R =   90.000 deg
};
P[923]{
   GP1:
	UF : 0, UT : 6,		CONFIG : 'N U T, 0, 0, 0',
	X =  41.934  mm,	Y =   -288.032  mm,	Z =   -248.111  mm,
	W =  90.000 deg,	P =   0.000 deg,	R =   90.000 deg
};
P[924]{
   GP1:
	UF : 0, UT : 6,		CONFIG : 'N U T, 0, 0, 0',
	X =  41.001  mm,	Y =   -288.556  mm,	Z =   -248.074  mm,
	W =  90.000 deg,	P =   0.000 deg,	R =   90.000 deg
};
P[925]{
   GP1:
	UF : 0, UT : 6,		CONFIG : 'N U T, 0, 0, 0',
	X =  34.964  mm,	Y =   -291.965  mm,	Z =   -247.887  mm,
	W =  90.000 deg,	P =   0.000 deg,	R =   90.000 deg
};
P[926]{
   GP1:
	UF : 0, UT : 6,		CONFIG : 'N U T, 0, 0, 0',
	X =  33.995  mm,	Y =   -292.584  mm,	Z =   -248.031  mm,
	W =  90.000 deg,	P =   0.000 deg,	R =   90.000 deg
};
P[927]{
   GP1:
	UF : 0, UT : 6,		CONFIG : 'N U T, 0, 0, 0',
	X =  31.669  mm,	Y =   -293.974  mm,	Z =   -248.147  mm,
	W =  90.000 deg,	P =   0.000 deg,	R =   90.000 deg
};
P[928]{
   GP1:
	UF : 0, UT : 6,		CONFIG : 'N U T, 0, 0, 0',
	X =  30.423  mm,	Y =   -294.534  mm,	Z =   -247.760  mm,
	W =  90.000 deg,	P =   0.000 deg,	R =   90.000 deg
};
P[929]{
   GP1:
	UF : 0, UT : 6,		CONFIG : 'N U T, 0, 0, 0',
	X =  29.568  mm,	Y =   -295.222  mm,	Z =   -248.232  mm,
	W =  90.000 deg,	P =   0.000 deg,	R =   90.000 deg
};
P[930]{
   GP1:
	UF : 0, UT : 6,		CONFIG : 'N U T, 0, 0, 0',
	X =  28.708  mm,	Y =   -295.618  mm,	Z =   -247.987  mm,
	W =  90.000 deg,	P =   0.000 deg,	R =   90.000 deg
};
P[931]{
   GP1:
	UF : 0, UT : 6,		CONFIG : 'N U T, 0, 0, 0',
	X =  25.014  mm,	Y =   -297.849  mm,	Z =   -248.225  mm,
	W =  90.000 deg,	P =   0.000 deg,	R =   90.000 deg
};
P[932]{
   GP1:
	UF : 0, UT : 6,		CONFIG : 'N U T, 0, 0, 0',
	X =  22.973  mm,	Y =   -299.018  mm,	Z =   -248.202  mm,
	W =  90.000 deg,	P =   0.000 deg,	R =   90.000 deg
};
P[933]{
   GP1:
	UF : 0, UT : 6,		CONFIG : 'N U T, 0, 0, 0',
	X =  21.933  mm,	Y =   -299.557  mm,	Z =   -248.054  mm,
	W =  90.000 deg,	P =   0.000 deg,	R =   90.000 deg
};
P[934]{
   GP1:
	UF : 0, UT : 6,		CONFIG : 'N U T, 0, 0, 0',
	X =  20.619  mm,	Y =   -300.399  mm,	Z =   -248.256  mm,
	W =  90.000 deg,	P =   0.000 deg,	R =   90.000 deg
};
P[935]{
   GP1:
	UF : 0, UT : 6,		CONFIG : 'N U T, 0, 0, 0',
	X =  19.451  mm,	Y =   -301.018  mm,	Z =   -248.123  mm,
	W =  90.000 deg,	P =   0.000 deg,	R =   90.000 deg
};
P[936]{
   GP1:
	UF : 0, UT : 6,		CONFIG : 'N U T, 0, 0, 0',
	X =  18.913  mm,	Y =   -301.327  mm,	Z =   -248.118  mm,
	W =  90.000 deg,	P =   0.000 deg,	R =   90.000 deg
};
P[937]{
   GP1:
	UF : 0, UT : 6,		CONFIG : 'N U T, 0, 0, 0',
	X =  17.580  mm,	Y =   -301.979  mm,	Z =   -247.829  mm,
	W =  90.000 deg,	P =   0.000 deg,	R =   90.000 deg
};
P[938]{
   GP1:
	UF : 0, UT : 6,		CONFIG : 'N U T, 0, 0, 0',
	X =  16.891  mm,	Y =   -302.377  mm,	Z =   -247.830  mm,
	W =  90.000 deg,	P =   0.000 deg,	R =   90.000 deg
};
P[939]{
   GP1:
	UF : 0, UT : 6,		CONFIG : 'N U T, 0, 0, 0',
	X =  15.958  mm,	Y =   -302.924  mm,	Z =   -247.853  mm,
	W =  90.000 deg,	P =   0.000 deg,	R =   90.000 deg
};
P[940]{
   GP1:
	UF : 0, UT : 6,		CONFIG : 'N U T, 0, 0, 0',
	X =  11.990  mm,	Y =   -305.363  mm,	Z =   -248.212  mm,
	W =  90.000 deg,	P =   0.000 deg,	R =   90.000 deg
};
P[941]{
   GP1:
	UF : 0, UT : 6,		CONFIG : 'N U T, 0, 0, 0',
	X =  10.914  mm,	Y =   -305.850  mm,	Z =   -247.885  mm,
	W =  90.000 deg,	P =   0.000 deg,	R =   90.000 deg
};
P[942]{
   GP1:
	UF : 0, UT : 6,		CONFIG : 'N U T, 0, 0, 0',
	X =  10.251  mm,	Y =   -306.301  mm,	Z =   -248.050  mm,
	W =  90.000 deg,	P =   0.000 deg,	R =   90.000 deg
};
P[943]{
   GP1:
	UF : 0, UT : 6,		CONFIG : 'N U T, 0, 0, 0',
	X =  9.370  mm,	Y =   -306.835  mm,	Z =   -248.112  mm,
	W =  90.000 deg,	P =   0.000 deg,	R =   90.000 deg
};
P[944]{
   GP1:
	UF : 0, UT : 6,		CONFIG : 'N U T, 0, 0, 0',
	X =  8.440  mm,	Y =   -307.330  mm,	Z =   -248.008  mm,
	W =  90.000 deg,	P =   0.000 deg,	R =   90.000 deg
};
P[945]{
   GP1:
	UF : 0, UT : 6,		CONFIG : 'N U T, 0, 0, 0',
	X =  7.502  mm,	Y =   -307.927  mm,	Z =   -248.145  mm,
	W =  90.000 deg,	P =   0.000 deg,	R =   90.000 deg
};
P[946]{
   GP1:
	UF : 0, UT : 6,		CONFIG : 'N U T, 0, 0, 0',
	X =  2.269  mm,	Y =   -310.902  mm,	Z =   -248.032  mm,
	W =  90.000 deg,	P =   0.000 deg,	R =   90.000 deg
};
P[947]{
   GP1:
	UF : 0, UT : 6,		CONFIG : 'N U T, 0, 0, 0',
	X =  1.125  mm,	Y =   -311.597  mm,	Z =   -248.117  mm,
	W =  90.000 deg,	P =   0.000 deg,	R =   90.000 deg
};
P[948]{
   GP1:
	UF : 0, UT : 6,		CONFIG : 'N U T, 0, 0, 0',
	X =  0.405  mm,	Y =   -311.997  mm,	Z =   -248.077  mm,
	W =  90.000 deg,	P =   0.000 deg,	R =   90.000 deg
};
P[949]{
   GP1:
	UF : 0, UT : 6,		CONFIG : 'N U T, 0, 0, 0',
	X =  -4.858  mm,	Y =   -315.078  mm,	Z =   -248.180  mm,
	W =  90.000 deg,	P =   0.000 deg,	R =   90.000 deg
};
P[950]{
   GP1:
	UF : 0, UT : 6,		CONFIG : 'N U T, 0, 0, 0',
	X =  -6.978  mm,	Y =   -316.220  mm,	Z =   -247.982  mm,
	W =  90.000 deg,	P =   0.000 deg,	R =   90.000 deg
};
P[951]{
   GP1:
	UF : 0, UT : 6,		CONFIG : 'N U T, 0, 0, 0',
	X =  -11.487  mm,	Y =   -318.920  mm,	Z =   -248.215  mm,
	W =  90.000 deg,	P =   0.000 deg,	R =   90.000 deg
};
P[952]{
   GP1:
	UF : 0, UT : 6,		CONFIG : 'N U T, 0, 0, 0',
	X =  -12.221  mm,	Y =   -319.284  mm,	Z =   -248.069  mm,
	W =  90.000 deg,	P =   0.000 deg,	R =   90.000 deg
};
P[953]{
   GP1:
	UF : 0, UT : 6,		CONFIG : 'N U T, 0, 0, 0',
	X =  -17.761  mm,	Y =   -322.375  mm,	Z =   -247.808  mm,
	W =  90.000 deg,	P =   0.000 deg,	R =   90.000 deg
};
P[954]{
   GP1:
	UF : 0, UT : 6,		CONFIG : 'N U T, 0, 0, 0',
	X =  -20.216  mm,	Y =   -323.821  mm,	Z =   -247.877  mm,
	W =  90.000 deg,	P =   0.000 deg,	R =   90.000 deg
};
P[955]{
   GP1:
	UF : 0, UT : 6,		CONFIG : 'N U T, 0, 0, 0',
	X =  -21.195  mm,	Y =   -324.463  mm,	Z =   -248.063  mm,
	W =  90.000 deg,	P =   0.000 deg,	R =   90.000 deg
};
P[956]{
   GP1:
	UF : 0, UT : 6,		CONFIG : 'N U T, 0, 0, 0',
	X =  -22.796  mm,	Y =   -325.302  mm,	Z =   -247.857  mm,
	W =  90.000 deg,	P =   0.000 deg,	R =   90.000 deg
};
P[957]{
   GP1:
	UF : 0, UT : 6,		CONFIG : 'N U T, 0, 0, 0',
	X =  -23.818  mm,	Y =   -326.004  mm,	Z =   -248.126  mm,
	W =  90.000 deg,	P =   0.000 deg,	R =   90.000 deg
};
P[958]{
   GP1:
	UF : 0, UT : 6,		CONFIG : 'N U T, 0, 0, 0',
	X =  -25.445  mm,	Y =   -326.809  mm,	Z =   -247.801  mm,
	W =  90.000 deg,	P =   0.000 deg,	R =   90.000 deg
};
P[959]{
   GP1:
	UF : 0, UT : 6,		CONFIG : 'N U T, 0, 0, 0',
	X =  -26.551  mm,	Y =   -327.575  mm,	Z =   -248.111  mm,
